LIN {X 0,Y 474.621,Z 246.364,A -85,B 0,C 180,E1 -7356.642,E2 -7356.642} C_VEL
LIN {X 0,Y 474.629,Z 246.359,A -85,B 0,C 180,E1 -7360.089,E2 -7360.089} C_VEL
LIN {X 0,Y 474.61,Z 246.369,A -85,B 0,C 180,E1 -7362.773,E2 -7362.773} C_VEL
LIN {X 0,Y 474.616,Z 246.361,A -85,B 0,C 180,E1 -7365.42,E2 -7365.42} C_VEL
LIN {X 0,Y 474.69,Z 246.352,A -85,B 0,C 180,E1 -7368.037,E2 -7368.037} C_VEL
LIN {X 0,Y 474.653,Z 246.356,A -85,B 0,C 180,E1 -7371.485,E2 -7371.485} C_VEL
LIN {X 0,Y 474.713,Z 246.35,A -85,B 0,C 180,E1 -7374.052,E2 -7374.052} C_VEL
LIN {X 0,Y 474.865,Z 246.329,A -85,B 0,C 180,E1 -7377.455,E2 -7377.455} C_VEL
LIN {X 0,Y 474.862,Z 246.332,A -85,B 0,C 180,E1 -7380,E2 -7380} C_VEL
LIN {X 0,Y 474.855,Z 246.338,A -85,B 0,C 180,E1 -7382.545,E2 -7382.545} C_VEL
LIN {X 0,Y 474.722,Z 246.349,A -85,B 0,C 180,E1 -7385.949,E2 -7385.949} C_VEL
LIN {X 0,Y 474.646,Z 246.363,A -85,B 0,C 180,E1 -7388.515,E2 -7388.515} C_VEL
LIN {X 0,Y 474.679,Z 246.356,A -85,B 0,C 180,E1 -7391.963,E2 -7391.963} C_VEL
LIN {X 0,Y 474.685,Z 246.352,A -85,B 0,C 180,E1 -7395.456,E2 -7395.456} C_VEL
LIN {X 0,Y 474.647,Z 246.356,A -85,B 0,C 180,E1 -7399.011,E2 -7399.011} C_VEL
LIN {X 0,Y 474.575,Z 246.368,A -85,B 0,C 180,E1 -7401.73,E2 -7401.73} C_VEL
LIN {X 0,Y 474.614,Z 246.364,A -85,B 0,C 180,E1 -7404.496,E2 -7404.496} C_VEL
LIN {X 0,Y 474.586,Z 246.364,A -85,B 0,C 180,E1 -7407.327,E2 -7407.327} C_VEL
LIN {X 0,Y 474.584,Z 246.369,A -85,B 0,C 180,E1 -7410.232,E2 -7410.232} C_VEL
LIN {X 0,Y 474.604,Z 246.362,A -85,B 0,C 180,E1 -7413.224,E2 -7413.224} C_VEL
LIN {X 0,Y 474.561,Z 246.37,A -85,B 0,C 180,E1 -7416.327,E2 -7416.327} C_VEL
LIN {X 0,Y 474.59,Z 246.367,A -85,B 0,C 180,E1 -7419.552,E2 -7419.552} C_VEL
LIN {X 0,Y 474.558,Z 246.367,A -85,B 0,C 180,E1 -7422.941,E2 -7422.941} C_VEL
LIN {X 0,Y 474.592,Z 246.369,A -85,B 0,C 180,E1 -7425.895,E2 -7425.895} C_VEL
LIN {X 0,Y 474.576,Z 246.366,A -85,B 0,C 180,E1 -7429.049,E2 -7429.049} C_VEL
LIN {X 0,Y 474.582,Z 246.372,A -85,B 0,C 180,E1 -7431.709,E2 -7431.709} C_VEL
LIN {X 0,Y 474.598,Z 246.362,A -85,B 0,C 180,E1 -7434.725,E2 -7434.725} C_VEL
LIN {X 0,Y 474.608,Z 246.366,A -85,B 0,C 180,E1 -7437.787,E2 -7437.787} C_VEL
LIN {X 0,Y 474.576,Z 246.366,A -85,B 0,C 180,E1 -7440.896,E2 -7440.896} C_VEL
LIN {X 0,Y 474.57,Z 246.372,A -85,B 0,C 180,E1 -7443.624,E2 -7443.624} C_VEL
LIN {X 0,Y 474.598,Z 246.363,A -85,B 0,C 180,E1 -7446.654,E2 -7446.654} C_VEL
LIN {X 0,Y 474.65,Z 246.362,A -85,B 0,C 180,E1 -7449.185,E2 -7449.185} C_VEL
LIN {X 0,Y 474.62,Z 246.363,A -85,B 0,C 180,E1 -7451.678,E2 -7451.678} C_VEL
LIN {X 0,Y 473.952,Z 246.443,A -85,B 0,C 180,E1 -7452.387,E2 -7452.387} C_VEL
LIN {X 0,Y 471.093,Z 246.804,A -85,B 0,C 180,E1 -7453.537,E2 -7453.537} C_VEL
LIN {X 0,Y 468.675,Z 247.109,A -85,B 0,C 180,E1 -7454.465,E2 -7454.465} C_VEL
LIN {X 0,Y 467.639,Z 247.236,A -85,B 0,C 180,E1 -7455.182,E2 -7455.182} C_VEL
LIN {X 0,Y 467.556,Z 247.244,A -85,B 0,C 180,E1 -7455.425,E2 -7455.425} C_VEL
LIN {X 0,Y 467.651,Z 247.231,A -85,B 0,C 180,E1 -7457.855,E2 -7457.855} C_VEL
LIN {X 0,Y 467.634,Z 247.345,A -85,B 0,C 180,E1 -7461.248,E2 -7461.248} C_VEL
LIN {X 0,Y 467.783,Z 248.185,A -85,B 0,C 180,E1 -7461.4,E2 -7461.4} C_VEL
LIN {X 0,Y 471.317,Z 258.187,A -85,B 0,C 180,E1 -7461.7,E2 -7461.7} C_VEL
LIN {X 0,Y 470.726,Z 335.625,A -85,B 0,C 180,E1 -7462.898,E2 -7462.898} C_VEL
LIN {X 0,Y 470.617,Z 348.645,A -85,B 0,C 180,E1 -7463.274,E2 -7463.274} C_VEL
LIN {X 0,Y 470.403,Z 361.714,A -85,B 0,C 180,E1 -7463.836,E2 -7463.836} C_VEL
LIN {X 0,Y 470.089,Z 373.512,A -85,B 0,C 180,E1 -7464.531,E2 -7464.531} C_VEL
LIN {X 0,Y 469.636,Z 384.793,A -85,B 0,C 180,E1 -7465.387,E2 -7465.387} C_VEL
LIN {X 0,Y 469.199,Z 394.954,A -85,B 0,C 180,E1 -7466.351,E2 -7466.351} C_VEL
LIN {X 0,Y 468.764,Z 404.111,A -85,B 0,C 180,E1 -7467.423,E2 -7467.423} C_VEL
LIN {X 0,Y 468.378,Z 412.945,A -85,B 0,C 180,E1 -7468.711,E2 -7468.711} C_VEL
LIN {X 0,Y 467.943,Z 420.099,A -85,B 0,C 180,E1 -7470,E2 -7470} C_VEL
LIN {X 0,Y 467.634,Z 425.83,A -85,B 0,C 180,E1 -7471.292,E2 -7471.292} C_VEL
LIN {X 0,Y 467.486,Z 430.339,A -85,B 0,C 180,E1 -7472.585,E2 -7472.585} C_VEL
LIN {X 0,Y 467.33,Z 432.748,A -85,B 0,C 180,E1 -7473.449,E2 -7473.449} C_VEL
LIN {X 0,Y 467.278,Z 436.248,A -85,B 0,C 180,E1 -7475.178,E2 -7475.178} C_VEL
LIN {X 0,Y 467.236,Z 437.399,A -85,B 0,C 180,E1 -7476.044,E2 -7476.044} C_VEL
LIN {X 0,Y 467.182,Z 438.465,A -85,B 0,C 180,E1 -7477.781,E2 -7477.781} C_VEL
LIN {X 0,Y 467.157,Z 438.436,A -85,B 0,C 180,E1 -7478.653,E2 -7478.653} C_VEL
LIN {X 0,Y 467.19,Z 438.007,A -85,B 0,C 180,E1 -7479.525,E2 -7479.525} C_VEL
LIN {X 0,Y 467.318,Z 435.892,A -85,B 0,C 180,E1 -7481.274,E2 -7481.274} C_VEL
LIN {X 0,Y 467.444,Z 433.216,A -85,B 0,C 180,E1 -7482.592,E2 -7482.592} C_VEL
LIN {X 0,Y 467.624,Z 429.5,A -85,B 0,C 180,E1 -7483.914,E2 -7483.914} C_VEL
LIN {X 0,Y 467.917,Z 424.627,A -85,B 0,C 180,E1 -7485.239,E2 -7485.239} C_VEL
LIN {X 0,Y 468.213,Z 418.444,A -85,B 0,C 180,E1 -7486.57,E2 -7486.57} C_VEL
LIN {X 0,Y 468.663,Z 410.633,A -85,B 0,C 180,E1 -7487.903,E2 -7487.903} C_VEL
LIN {X 0,Y 469.116,Z 402.581,A -85,B 0,C 180,E1 -7489.017,E2 -7489.017} C_VEL
LIN {X 0,Y 469.568,Z 392.679,A -85,B 0,C 180,E1 -7490.135,E2 -7490.135} C_VEL
LIN {X 0,Y 469.997,Z 382.87,A -85,B 0,C 180,E1 -7491.031,E2 -7491.031} C_VEL
LIN {X 0,Y 470.489,Z 372.14,A -85,B 0,C 180,E1 -7491.813,E2 -7491.813} C_VEL
LIN {X 0,Y 470.802,Z 360.376,A -85,B 0,C 180,E1 -7492.482,E2 -7492.482} C_VEL
LIN {X 0,Y 470.994,Z 347.261,A -85,B 0,C 180,E1 -7493.031,E2 -7493.031} C_VEL
LIN {X 0,Y 471.146,Z 334.596,A -85,B 0,C 180,E1 -7493.372,E2 -7493.372} C_VEL
LIN {X 0,Y 471.661,Z 258.296,A -85,B 0,C 180,E1 -7494.57,E2 -7494.57} C_VEL
LIN {X 0,Y 467.796,Z 248.157,A -85,B 0,C 180,E1 -7494.925,E2 -7494.925} C_VEL
LIN {X 0,Y 467.618,Z 247.318,A -85,B 0,C 180,E1 -7495.096,E2 -7495.096} C_VEL
LIN {X 0,Y 467.564,Z 247.242,A -85,B 0,C 180,E1 -7497.772,E2 -7497.772} C_VEL
LIN {X 0,Y 467.552,Z 247.228,A -85,B 0,C 180,E1 -7501.041,E2 -7501.041} C_VEL
LIN {X 0,Y 467.577,Z 247.243,A -85,B 0,C 180,E1 -7504.239,E2 -7504.239} C_VEL
LIN {X 0,Y 467.535,Z 247.227,A -85,B 0,C 180,E1 -7507.183,E2 -7507.183} C_VEL
LIN {X 0,Y 467.556,Z 247.246,A -85,B 0,C 180,E1 -7510.266,E2 -7510.266} C_VEL
LIN {X 0,Y 467.545,Z 247.243,A -85,B 0,C 180,E1 -7513.745,E2 -7513.745} C_VEL
LIN {X 0,Y 467.542,Z 247.241,A -85,B 0,C 180,E1 -7516.253,E2 -7516.253} C_VEL
LIN {X 0,Y 467.554,Z 247.242,A -85,B 0,C 180,E1 -7519.732,E2 -7519.732} C_VEL
LIN {X 0,Y 467.514,Z 247.239,A -85,B 0,C 180,E1 -7522.818,E2 -7522.818} C_VEL
LIN {X 0,Y 467.583,Z 247.24,A -85,B 0,C 180,E1 -7525.758,E2 -7525.758} C_VEL
LIN {X 0,Y 467.563,Z 247.226,A -85,B 0,C 180,E1 -7528.955,E2 -7528.955} C_VEL
LIN {X 0,Y 467.542,Z 247.245,A -85,B 0,C 180,E1 -7532.226,E2 -7532.226} C_VEL
LIN {X 0,Y 467.564,Z 247.238,A -85,B 0,C 180,E1 -7535.11,E2 -7535.11} C_VEL
LIN {X 0,Y 467.528,Z 247.228,A -85,B 0,C 180,E1 -7537.925,E2 -7537.925} C_VEL
LIN {X 0,Y 467.615,Z 247.23,A -85,B 0,C 180,E1 -7540.692,E2 -7540.692} C_VEL
LIN {X 0,Y 467.631,Z 247.23,A -85,B 0,C 180,E1 -7544.304,E2 -7544.304} C_VEL
LIN {X 0,Y 467.649,Z 247.235,A -85,B 0,C 180,E1 -7547.854,E2 -7547.854} C_VEL
LIN {X 0,Y 467.649,Z 247.224,A -85,B 0,C 180,E1 -7551.356,E2 -7551.356} C_VEL
LIN {X 0,Y 467.694,Z 247.227,A -85,B 0,C 180,E1 -7553.962,E2 -7553.962} C_VEL
LIN {X 0,Y 467.804,Z 247.209,A -85,B 0,C 180,E1 -7557.417,E2 -7557.417} C_VEL
LIN {X 0,Y 467.839,Z 247.206,A -85,B 0,C 180,E1 -7560,E2 -7560} C_VEL
LIN {X 0,Y 467.813,Z 247.204,A -85,B 0,C 180,E1 -7562.583,E2 -7562.583} C_VEL
LIN {X 0,Y 467.685,Z 247.223,A -85,B 0,C 180,E1 -7566.038,E2 -7566.038} C_VEL
LIN {X 0,Y 467.657,Z 247.224,A -85,B 0,C 180,E1 -7568.643,E2 -7568.643} C_VEL
LIN {X 0,Y 467.646,Z 247.225,A -85,B 0,C 180,E1 -7572.357,E2 -7572.357} C_VEL
LIN {X 0,Y 467.616,Z 247.235,A -85,B 0,C 180,E1 -7575.873,E2 -7575.873} C_VEL
LIN {X 0,Y 467.612,Z 247.239,A -85,B 0,C 180,E1 -7579.308,E2 -7579.308} C_VEL
LIN {X 0,Y 467.523,Z 247.242,A -85,B 0,C 180,E1 -7582.074,E2 -7582.074} C_VEL
LIN {X 0,Y 467.548,Z 247.246,A -85,B 0,C 180,E1 -7584.89,E2 -7584.89} C_VEL
LIN {X 0,Y 467.536,Z 247.235,A -85,B 0,C 180,E1 -7587.774,E2 -7587.774} C_VEL
LIN {X 0,Y 467.531,Z 247.251,A -85,B 0,C 180,E1 -7591.039,E2 -7591.039} C_VEL
LIN {X 0,Y 467.562,Z 247.232,A -85,B 0,C 180,E1 -7593.79,E2 -7593.79} C_VEL
LIN {X 0,Y 467.5,Z 247.254,A -85,B 0,C 180,E1 -7596.965,E2 -7596.965} C_VEL
LIN {X 0,Y 467.556,Z 247.24,A -85,B 0,C 180,E1 -7599.952,E2 -7599.952} C_VEL
LIN {X 0,Y 467.513,Z 247.25,A -85,B 0,C 180,E1 -7602.569,E2 -7602.569} C_VEL
LIN {X 0,Y 467.558,Z 247.245,A -85,B 0,C 180,E1 -7605.052,E2 -7605.052} C_VEL
LIN {X 0,Y 467.551,Z 247.245,A -85,B 0,C 180,E1 -7608.727,E2 -7608.727} C_VEL
LIN {X 0,Y 467.531,Z 247.242,A -85,B 0,C 180,E1 -7611.953,E2 -7611.953} C_VEL
LIN {X 0,Y 467.547,Z 247.237,A -85,B 0,C 180,E1 -7615.166,E2 -7615.166} C_VEL
LIN {X 0,Y 467.544,Z 247.239,A -85,B 0,C 180,E1 -7618.257,E2 -7618.257} C_VEL
LIN {X 0,Y 467.564,Z 247.452,A -85,B 0,C 180,E1 -7620.587,E2 -7620.587} C_VEL
LIN {X 0,Y 470.411,Z 260.504,A -85,B 0,C 180,E1 -7622.651,E2 -7622.651} C_VEL
LIN {X 0,Y 470.807,Z 263.899,A -85,B 0,C 180,E1 -7623.157,E2 -7623.157} C_VEL
LIN {X 0,Y 469.848,Z 285.592,A -85,B 0,C 180,E1 -7626.18,E2 -7626.18} C_VEL
LIN {X 0,Y 469.068,Z 307.215,A -85,B 0,C 180,E1 -7629.155,E2 -7629.155} C_VEL
LIN {X 0,Y 468.414,Z 328.784,A -85,B 0,C 180,E1 -7632.087,E2 -7632.087} C_VEL
LIN {X 0,Y 468.237,Z 334.47,A -85,B 0,C 180,E1 -7632.84,E2 -7632.84} C_VEL
LIN {X 0,Y 470.969,Z 358.48,A -85,B 0,C 180,E1 -7633.353,E2 -7633.353} C_VEL
LIN {X 0,Y 471.032,Z 374.98,A -85,B 0,C 180,E1 -7633.615,E2 -7633.615} C_VEL
LIN {X 0,Y 470.493,Z 444.897,A -85,B 0,C 180,E1 -7634.708,E2 -7634.708} C_VEL
LIN {X 0,Y 470.06,Z 458.205,A -85,B 0,C 180,E1 -7635.082,E2 -7635.082} C_VEL
LIN {X 0,Y 469.548,Z 470.424,A -85,B 0,C 180,E1 -7635.591,E2 -7635.591} C_VEL
LIN {X 0,Y 469.037,Z 481.969,A -85,B 0,C 180,E1 -7636.239,E2 -7636.239} C_VEL
LIN {X 0,Y 468.504,Z 492.547,A -85,B 0,C 180,E1 -7636.996,E2 -7636.996} C_VEL
LIN {X 0,Y 468.07,Z 503.465,A -85,B 0,C 180,E1 -7637.975,E2 -7637.975} C_VEL
LIN {X 0,Y 467.631,Z 512.407,A -85,B 0,C 180,E1 -7638.953,E2 -7638.953} C_VEL
LIN {X 0,Y 467.222,Z 522.165,A -85,B 0,C 180,E1 -7640.257,E2 -7640.257} C_VEL
LIN {X 0,Y 467.016,Z 529.966,A -85,B 0,C 180,E1 -7641.563,E2 -7641.563} C_VEL
LIN {X 0,Y 466.912,Z 537.197,A -85,B 0,C 180,E1 -7643.084,E2 -7643.084} C_VEL
LIN {X 0,Y 466.899,Z 542.022,A -85,B 0,C 180,E1 -7644.385,E2 -7644.385} C_VEL
LIN {X 0,Y 466.948,Z 545.721,A -85,B 0,C 180,E1 -7645.684,E2 -7645.684} C_VEL
LIN {X 0,Y 466.99,Z 547.631,A -85,B 0,C 180,E1 -7646.549,E2 -7646.549} C_VEL
LIN {X 0,Y 466.887,Z 550.075,A -85,B 0,C 180,E1 -7648.274,E2 -7648.274} C_VEL
LIN {X 0,Y 466.897,Z 550.703,A -85,B 0,C 180,E1 -7649.137,E2 -7649.137} C_VEL
LIN {X 0,Y 466.917,Z 550.927,A -85,B 0,C 180,E1 -7650,E2 -7650} C_VEL
LIN {X 0,Y 466.897,Z 550.703,A -85,B 0,C 180,E1 -7650.862,E2 -7650.862} C_VEL
LIN {X 0,Y 466.91,Z 549.066,A -85,B 0,C 180,E1 -7652.588,E2 -7652.588} C_VEL
LIN {X 0,Y 466.987,Z 547.639,A -85,B 0,C 180,E1 -7653.451,E2 -7653.451} C_VEL
LIN {X 0,Y 466.887,Z 544.613,A -85,B 0,C 180,E1 -7654.749,E2 -7654.749} C_VEL
LIN {X 0,Y 466.888,Z 539.767,A -85,B 0,C 180,E1 -7656.251,E2 -7656.251} C_VEL
LIN {X 0,Y 466.974,Z 533.211,A -85,B 0,C 180,E1 -7657.784,E2 -7657.784} C_VEL
LIN {X 0,Y 467.139,Z 526.131,A -85,B 0,C 180,E1 -7659.089,E2 -7659.089} C_VEL
LIN {X 0,Y 467.403,Z 517.268,A -85,B 0,C 180,E1 -7660.395,E2 -7660.395} C_VEL
LIN {X 0,Y 467.757,Z 507.203,A -85,B 0,C 180,E1 -7661.592,E2 -7661.592} C_VEL
LIN {X 0,Y 468.289,Z 497.301,A -85,B 0,C 180,E1 -7662.547,E2 -7662.547} C_VEL
LIN {X 0,Y 468.754,Z 485.756,A -85,B 0,C 180,E1 -7663.437,E2 -7663.437} C_VEL
LIN {X 0,Y 469.301,Z 473.12,A -85,B 0,C 180,E1 -7664.194,E2 -7664.194} C_VEL
LIN {X 0,Y 469.808,Z 460.235,A -85,B 0,C 180,E1 -7664.76,E2 -7664.76} C_VEL
LIN {X 0,Y 470.254,Z 446.5,A -85,B 0,C 180,E1 -7665.161,E2 -7665.161} C_VEL
LIN {X 0,Y 470.591,Z 400.642,A -85,B 0,C 180,E1 -7665.886,E2 -7665.886} C_VEL
LIN {X 0,Y 470.806,Z 359,A -85,B 0,C 180,E1 -7666.521,E2 -7666.521} C_VEL
LIN {X 0,Y 468.174,Z 335.117,A -85,B 0,C 180,E1 -7666.992,E2 -7666.992} C_VEL
LIN {X 0,Y 468.811,Z 312.964,A -85,B 0,C 180,E1 -7669.94,E2 -7669.94} C_VEL
LIN {X 0,Y 469.582,Z 287.643,A -85,B 0,C 180,E1 -7673.366,E2 -7673.366} C_VEL
LIN {X 0,Y 470.464,Z 263.767,A -85,B 0,C 180,E1 -7676.624,E2 -7676.624} C_VEL
LIN {X 0,Y 469.895,Z 258.487,A -85,B 0,C 180,E1 -7677.38,E2 -7677.38} C_VEL
LIN {X 0,Y 467.548,Z 247.389,A -85,B 0,C 180,E1 -7679.076,E2 -7679.076} C_VEL
LIN {X 0,Y 467.541,Z 247.249,A -85,B 0,C 180,E1 -7681.742,E2 -7681.742} C_VEL
LIN {X 0,Y 467.544,Z 247.245,A -85,B 0,C 180,E1 -7684.833,E2 -7684.833} C_VEL
LIN {X 0,Y 467.528,Z 247.244,A -85,B 0,C 180,E1 -7688.047,E2 -7688.047} C_VEL
LIN {X 0,Y 467.547,Z 247.248,A -85,B 0,C 180,E1 -7691.404,E2 -7691.404} C_VEL
LIN {X 0,Y 467.553,Z 247.245,A -85,B 0,C 180,E1 -7695.051,E2 -7695.051} C_VEL
LIN {X 0,Y 467.551,Z 247.243,A -85,B 0,C 180,E1 -7698.725,E2 -7698.725} C_VEL
LIN {X 0,Y 467.534,Z 247.243,A -85,B 0,C 180,E1 -7701.952,E2 -7701.952} C_VEL
LIN {X 0,Y 467.535,Z 247.249,A -85,B 0,C 180,E1 -7705.165,E2 -7705.165} C_VEL
LIN {X 0,Y 467.533,Z 247.243,A -85,B 0,C 180,E1 -7708.256,E2 -7708.256} C_VEL
LIN {X 0,Y 467.527,Z 247.248,A -85,B 0,C 180,E1 -7711.247,E2 -7711.247} C_VEL
LIN {X 0,Y 467.549,Z 247.242,A -85,B 0,C 180,E1 -7714.405,E2 -7714.405} C_VEL
LIN {X 0,Y 467.558,Z 247.246,A -85,B 0,C 180,E1 -7716.995,E2 -7716.995} C_VEL
LIN {X 0,Y 467.598,Z 247.234,A -85,B 0,C 180,E1 -7719.776,E2 -7719.776} C_VEL
LIN {X 0,Y 467.573,Z 247.242,A -85,B 0,C 180,E1 -7722.505,E2 -7722.505} C_VEL
LIN {X 0,Y 467.578,Z 247.239,A -85,B 0,C 180,E1 -7725.196,E2 -7725.196} C_VEL
LIN {X 0,Y 467.642,Z 247.229,A -85,B 0,C 180,E1 -7727.854,E2 -7727.854} C_VEL
LIN {X 0,Y 467.621,Z 247.232,A -85,B 0,C 180,E1 -7731.356,E2 -7731.356} C_VEL
LIN {X 0,Y 467.678,Z 247.225,A -85,B 0,C 180,E1 -7733.962,E2 -7733.962} C_VEL
LIN {X 0,Y 467.806,Z 247.208,A -85,B 0,C 180,E1 -7737.417,E2 -7737.417} C_VEL
LIN {X 0,Y 467.832,Z 247.207,A -85,B 0,C 180,E1 -7740,E2 -7740} C_VEL
LIN {X 0,Y 467.795,Z 247.216,A -85,B 0,C 180,E1 -7742.583,E2 -7742.583} C_VEL
LIN {X 0,Y 467.687,Z 247.227,A -85,B 0,C 180,E1 -7746.038,E2 -7746.038} C_VEL
LIN {X 0,Y 467.615,Z 247.237,A -85,B 0,C 180,E1 -7748.644,E2 -7748.644} C_VEL
LIN {X 0,Y 467.635,Z 247.237,A -85,B 0,C 180,E1 -7752.354,E2 -7752.354} C_VEL
LIN {X 0,Y 467.611,Z 247.236,A -85,B 0,C 180,E1 -7755.874,E2 -7755.874} C_VEL
LIN {X 0,Y 467.606,Z 247.233,A -85,B 0,C 180,E1 -7759.309,E2 -7759.309} C_VEL
LIN {X 0,Y 467.519,Z 247.252,A -85,B 0,C 180,E1 -7762.075,E2 -7762.075} C_VEL
LIN {X 0,Y 467.543,Z 247.241,A -85,B 0,C 180,E1 -7764.891,E2 -7764.891} C_VEL
LIN {X 0,Y 467.533,Z 247.247,A -85,B 0,C 180,E1 -7767.775,E2 -7767.775} C_VEL
LIN {X 0,Y 467.535,Z 247.242,A -85,B 0,C 180,E1 -7771.041,E2 -7771.041} C_VEL
LIN {X 0,Y 467.566,Z 247.242,A -85,B 0,C 180,E1 -7774.241,E2 -7774.241} C_VEL
LIN {X 0,Y 467.505,Z 247.247,A -85,B 0,C 180,E1 -7777.182,E2 -7777.182} C_VEL
LIN {X 0,Y 467.509,Z 247.248,A -85,B 0,C 180,E1 -7780.272,E2 -7780.272} C_VEL
LIN {X 0,Y 467.509,Z 247.246,A -85,B 0,C 180,E1 -7782.57,E2 -7782.57} C_VEL
LIN {X 0,Y 467.556,Z 247.24,A -85,B 0,C 180,E1 -7785.053,E2 -7785.053} C_VEL
LIN {X 0,Y 467.545,Z 247.241,A -85,B 0,C 180,E1 -7788.729,E2 -7788.729} C_VEL
LIN {X 0,Y 467.533,Z 247.246,A -85,B 0,C 180,E1 -7791.954,E2 -7791.954} C_VEL
LIN {X 0,Y 467.536,Z 247.245,A -85,B 0,C 180,E1 -7795.166,E2 -7795.166} C_VEL
LIN {X 0,Y 467.54,Z 247.242,A -85,B 0,C 180,E1 -7798.258,E2 -7798.258} C_VEL
LIN {X 0,Y 467.525,Z 247.248,A -85,B 0,C 180,E1 -7801.248,E2 -7801.248} C_VEL
LIN {X 0,Y 467.561,Z 247.239,A -85,B 0,C 180,E1 -7804.406,E2 -7804.406} C_VEL
LIN {X 0,Y 467.552,Z 247.243,A -85,B 0,C 180,E1 -7806.996,E2 -7806.996} C_VEL
LIN {X 0,Y 467.594,Z 247.238,A -85,B 0,C 180,E1 -7809.777,E2 -7809.777} C_VEL
LIN {X 0,Y 467.577,Z 247.237,A -85,B 0,C 180,E1 -7812.506,E2 -7812.506} C_VEL
LIN {X 0,Y 467.556,Z 247.244,A -85,B 0,C 180,E1 -7815.425,E2 -7815.425} C_VEL
LIN {X 0,Y 466.897,Z 247.323,A -85,B 0,C 180,E1 -7816.144,E2 -7816.144} C_VEL
LIN {X 0,Y 464.065,Z 247.682,A -85,B 0,C 180,E1 -7817.313,E2 -7817.313} C_VEL
LIN {X 0,Y 461.667,Z 247.978,A -85,B 0,C 180,E1 -7818.256,E2 -7818.256} C_VEL
LIN {X 0,Y 460.634,Z 248.109,A -85,B 0,C 180,E1 -7818.984,E2 -7818.984} C_VEL
LIN {X 0,Y 460.549,Z 248.116,A -85,B 0,C 180,E1 -7819.23,E2 -7819.23} C_VEL
LIN {X 0,Y 460.608,Z 248.343,A -85,B 0,C 180,E1 -7821.058,E2 -7821.058} C_VEL
LIN {X 0,Y 460.859,Z 249.412,A -85,B 0,C 180,E1 -7821.191,E2 -7821.191} C_VEL
LIN {X 0,Y 464.461,Z 259.967,A -85,B 0,C 180,E1 -7821.494,E2 -7821.494} C_VEL
LIN {X 0,Y 463.859,Z 337.152,A -85,B 0,C 180,E1 -7822.711,E2 -7822.711} C_VEL
LIN {X 0,Y 463.781,Z 350.665,A -85,B 0,C 180,E1 -7823.119,E2 -7823.119} C_VEL
LIN {X 0,Y 463.526,Z 362.345,A -85,B 0,C 180,E1 -7823.635,E2 -7823.635} C_VEL
LIN {X 0,Y 463.205,Z 374.206,A -85,B 0,C 180,E1 -7824.341,E2 -7824.341} C_VEL
LIN {X 0,Y 462.731,Z 385.516,A -85,B 0,C 180,E1 -7825.209,E2 -7825.209} C_VEL
LIN {X 0,Y 462.269,Z 395.701,A -85,B 0,C 180,E1 -7826.187,E2 -7826.187} C_VEL
LIN {X 0,Y 461.87,Z 404.033,A -85,B 0,C 180,E1 -7827.166,E2 -7827.166} C_VEL
LIN {X 0,Y 461.479,Z 411.725,A -85,B 0,C 180,E1 -7828.255,E2 -7828.255} C_VEL
LIN {X 0,Y 461.029,Z 419.262,A -85,B 0,C 180,E1 -7829.564,E2 -7829.564} C_VEL
LIN {X 0,Y 460.704,Z 425.308,A -85,B 0,C 180,E1 -7830.874,E2 -7830.874} C_VEL
LIN {X 0,Y 460.484,Z 430.114,A -85,B 0,C 180,E1 -7832.187,E2 -7832.187} C_VEL
LIN {X 0,Y 460.283,Z 433.835,A -85,B 0,C 180,E1 -7833.502,E2 -7833.502} C_VEL
LIN {X 0,Y 460.248,Z 435.748,A -85,B 0,C 180,E1 -7834.379,E2 -7834.379} C_VEL
LIN {X 0,Y 460.234,Z 437.259,A -85,B 0,C 180,E1 -7835.257,E2 -7835.257} C_VEL
LIN {X 0,Y 460.166,Z 438.963,A -85,B 0,C 180,E1 -7836.909,E2 -7836.909} C_VEL
LIN {X 0,Y 460.142,Z 439.334,A -85,B 0,C 180,E1 -7837.901,E2 -7837.901} C_VEL
LIN {X 0,Y 460.125,Z 439.267,A -85,B 0,C 180,E1 -7838.786,E2 -7838.786} C_VEL
LIN {X 0,Y 460.141,Z 438.769,A -85,B 0,C 180,E1 -7839.672,E2 -7839.672} C_VEL
LIN {X 0,Y 460.307,Z 436.579,A -85,B 0,C 180,E1 -7841.448,E2 -7841.448} C_VEL
LIN {X 0,Y 460.433,Z 433.827,A -85,B 0,C 180,E1 -7842.787,E2 -7842.787} C_VEL
LIN {X 0,Y 460.654,Z 430.029,A -85,B 0,C 180,E1 -7844.129,E2 -7844.129} C_VEL
LIN {X 0,Y 460.99,Z 425.067,A -85,B 0,C 180,E1 -7845.474,E2 -7845.474} C_VEL
LIN {X 0,Y 461.305,Z 418.775,A -85,B 0,C 180,E1 -7846.826,E2 -7846.826} C_VEL
LIN {X 0,Y 461.816,Z 410.809,A -85,B 0,C 180,E1 -7848.178,E2 -7848.178} C_VEL
LIN {X 0,Y 462.329,Z 402.049,A -85,B 0,C 180,E1 -7849.381,E2 -7849.381} C_VEL
LIN {X 0,Y 462.759,Z 392.55,A -85,B 0,C 180,E1 -7850.445,E2 -7850.445} C_VEL
LIN {X 0,Y 463.24,Z 382.457,A -85,B 0,C 180,E1 -7851.353,E2 -7851.353} C_VEL
LIN {X 0,Y 463.772,Z 371.385,A -85,B 0,C 180,E1 -7852.145,E2 -7852.145} C_VEL
LIN {X 0,Y 464.081,Z 359.466,A -85,B 0,C 180,E1 -7852.81,E2 -7852.81} C_VEL
LIN {X 0,Y 464.273,Z 346.755,A -85,B 0,C 180,E1 -7853.325,E2 -7853.325} C_VEL
LIN {X 0,Y 464.431,Z 333.014,A -85,B 0,C 180,E1 -7853.671,E2 -7853.671} C_VEL
LIN {X 0,Y 464.952,Z 259.822,A -85,B 0,C 180,E1 -7854.832,E2 -7854.832} C_VEL
LIN {X 0,Y 460.76,Z 249.177,A -85,B 0,C 180,E1 -7855.21,E2 -7855.21} C_VEL
LIN {X 0,Y 460.555,Z 248.238,A -85,B 0,C 180,E1 -7855.373,E2 -7855.373} C_VEL
LIN {X 0,Y 460.518,Z 248.119,A -85,B 0,C 180,E1 -7858.235,E2 -7858.235} C_VEL
LIN {X 0,Y 460.522,Z 248.104,A -85,B 0,C 180,E1 -7861.282,E2 -7861.282} C_VEL
LIN {X 0,Y 460.522,Z 248.116,A -85,B 0,C 180,E1 -7864.503,E2 -7864.503} C_VEL
LIN {X 0,Y 460.493,Z 248.11,A -85,B 0,C 180,E1 -7867.623,E2 -7867.623} C_VEL
LIN {X 0,Y 460.515,Z 248.117,A -85,B 0,C 180,E1 -7871.012,E2 -7871.012} C_VEL
LIN {X 0,Y 460.51,Z 248.125,A -85,B 0,C 180,E1 -7874.589,E2 -7874.589} C_VEL
LIN {X 0,Y 460.472,Z 248.118,A -85,B 0,C 180,E1 -7877.812,E2 -7877.812} C_VEL
LIN {X 0,Y 460.508,Z 248.123,A -85,B 0,C 180,E1 -7880.135,E2 -7880.135} C_VEL
LIN {X 0,Y 460.458,Z 248.117,A -85,B 0,C 180,E1 -7883.468,E2 -7883.468} C_VEL
LIN {X 0,Y 460.524,Z 248.118,A -85,B 0,C 180,E1 -7886.674,E2 -7886.674} C_VEL
LIN {X 0,Y 460.502,Z 248.105,A -85,B 0,C 180,E1 -7889.759,E2 -7889.759} C_VEL
LIN {X 0,Y 460.487,Z 248.124,A -85,B 0,C 180,E1 -7892.75,E2 -7892.75} C_VEL
LIN {X 0,Y 460.517,Z 248.118,A -85,B 0,C 180,E1 -7895.666,E2 -7895.666} C_VEL
LIN {X 0,Y 460.516,Z 248.101,A -85,B 0,C 180,E1 -7898.578,E2 -7898.578} C_VEL
LIN {X 0,Y 460.578,Z 248.107,A -85,B 0,C 180,E1 -7901.31,E2 -7901.31} C_VEL
LIN {X 0,Y 460.599,Z 248.11,A -85,B 0,C 180,E1 -7904.058,E2 -7904.058} C_VEL
LIN {X 0,Y 460.602,Z 248.11,A -85,B 0,C 180,E1 -7907.665,E2 -7907.665} C_VEL
LIN {X 0,Y 460.601,Z 248.101,A -85,B 0,C 180,E1 -7911.223,E2 -7911.223} C_VEL
LIN {X 0,Y 460.66,Z 248.104,A -85,B 0,C 180,E1 -7913.869,E2 -7913.869} C_VEL
LIN {X 0,Y 460.748,Z 248.087,A -85,B 0,C 180,E1 -7917.377,E2 -7917.377} C_VEL
LIN {X 0,Y 460.809,Z 248.082,A -85,B 0,C 180,E1 -7920,E2 -7920} C_VEL
LIN {X 0,Y 460.758,Z 248.083,A -85,B 0,C 180,E1 -7922.623,E2 -7922.623} C_VEL
LIN {X 0,Y 460.651,Z 248.098,A -85,B 0,C 180,E1 -7926.131,E2 -7926.131} C_VEL
LIN {X 0,Y 460.608,Z 248.103,A -85,B 0,C 180,E1 -7928.776,E2 -7928.776} C_VEL
LIN {X 0,Y 460.59,Z 248.104,A -85,B 0,C 180,E1 -7932.435,E2 -7932.435} C_VEL
LIN {X 0,Y 460.572,Z 248.112,A -85,B 0,C 180,E1 -7935.988,E2 -7935.988} C_VEL
LIN {X 0,Y 460.558,Z 248.112,A -85,B 0,C 180,E1 -7938.899,E2 -7938.899} C_VEL
LIN {X 0,Y 460.509,Z 248.12,A -85,B 0,C 180,E1 -7941.486,E2 -7941.486} C_VEL
LIN {X 0,Y 460.509,Z 248.119,A -85,B 0,C 180,E1 -7944.334,E2 -7944.334} C_VEL
LIN {X 0,Y 460.482,Z 248.114,A -85,B 0,C 180,E1 -7947.25,E2 -7947.25} C_VEL
LIN {X 0,Y 460.487,Z 248.121,A -85,B 0,C 180,E1 -7950.242,E2 -7950.242} C_VEL
LIN {X 0,Y 460.512,Z 248.112,A -85,B 0,C 180,E1 -7953.326,E2 -7953.326} C_VEL
LIN {X 0,Y 460.455,Z 248.128,A -85,B 0,C 180,E1 -7956.531,E2 -7956.531} C_VEL
LIN {X 0,Y 460.505,Z 248.118,A -85,B 0,C 180,E1 -7959.865,E2 -7959.865} C_VEL
LIN {X 0,Y 460.452,Z 248.126,A -85,B 0,C 180,E1 -7962.893,E2 -7962.893} C_VEL
LIN {X 0,Y 460.5,Z 248.119,A -85,B 0,C 180,E1 -7965.832,E2 -7965.832} C_VEL
LIN {X 0,Y 460.504,Z 248.119,A -85,B 0,C 180,E1 -7968.986,E2 -7968.986} C_VEL
LIN {X 0,Y 460.476,Z 248.124,A -85,B 0,C 180,E1 -7972.375,E2 -7972.375} C_VEL
LIN {X 0,Y 460.531,Z 248.114,A -85,B 0,C 180,E1 -7975.623,E2 -7975.623} C_VEL
LIN {X 0,Y 460.503,Z 248.12,A -85,B 0,C 180,E1 -7978.742,E2 -7978.742} C_VEL
LIN {X 0,Y 460.526,Z 248.315,A -85,B 0,C 180,E1 -7980.319,E2 -7980.319} C_VEL
LIN {X 0,Y 463.436,Z 261.52,A -85,B 0,C 180,E1 -7982.45,E2 -7982.45} C_VEL
LIN {X 0,Y 463.905,Z 264.918,A -85,B 0,C 180,E1 -7982.968,E2 -7982.968} C_VEL
LIN {X 0,Y 462.923,Z 286.594,A -85,B 0,C 180,E1 -7986.039,E2 -7986.039} C_VEL
LIN {X 0,Y 462.094,Z 308.192,A -85,B 0,C 180,E1 -7989.059,E2 -7989.059} C_VEL
LIN {X 0,Y 461.316,Z 331.385,A -85,B 0,C 180,E1 -7992.26,E2 -7992.26} C_VEL
LIN {X 0,Y 461.279,Z 333.981,A -85,B 0,C 180,E1 -7992.568,E2 -7992.568} C_VEL
LIN {X 0,Y 464.071,Z 357.869,A -85,B 0,C 180,E1 -7993.076,E2 -7993.076} C_VEL
LIN {X 0,Y 464.375,Z 364.598,A -85,B 0,C 180,E1 -7993.195,E2 -7993.195} C_VEL
LIN {X 0,Y 463.652,Z 444.972,A -85,B 0,C 180,E1 -7994.477,E2 -7994.477} C_VEL
LIN {X 0,Y 463.178,Z 458.722,A -85,B 0,C 180,E1 -7994.883,E2 -7994.883} C_VEL
LIN {X 0,Y 462.668,Z 470.01,A -85,B 0,C 180,E1 -7995.372,E2 -7995.372} C_VEL
LIN {X 0,Y 462.121,Z 481.434,A -85,B 0,C 180,E1 -7996.029,E2 -7996.029} C_VEL
LIN {X 0,Y 461.47,Z 493.521,A -85,B 0,C 180,E1 -7996.931,E2 -7996.931} C_VEL
LIN {X 0,Y 461.023,Z 503.875,A -85,B 0,C 180,E1 -7997.9,E2 -7997.9} C_VEL
LIN {X 0,Y 460.517,Z 513.5,A -85,B 0,C 180,E1 -7999.003,E2 -7999.003} C_VEL
LIN {X 0,Y 460.104,Z 522.802,A -85,B 0,C 180,E1 -8000.327,E2 -8000.327} C_VEL
LIN {X 0,Y 459.931,Z 530.333,A -85,B 0,C 180,E1 -8001.653,E2 -8001.653} C_VEL
LIN {X 0,Y 459.845,Z 536.404,A -85,B 0,C 180,E1 -8002.977,E2 -8002.977} C_VEL
LIN {X 0,Y 459.829,Z 541.214,A -85,B 0,C 180,E1 -8004.298,E2 -8004.298} C_VEL
LIN {X 0,Y 459.888,Z 544.902,A -85,B 0,C 180,E1 -8005.617,E2 -8005.617} C_VEL
LIN {X 0,Y 459.941,Z 546.804,A -85,B 0,C 180,E1 -8006.496,E2 -8006.496} C_VEL
LIN {X 0,Y 459.832,Z 549.237,A -85,B 0,C 180,E1 -8008.248,E2 -8008.248} C_VEL
LIN {X 0,Y 459.844,Z 549.861,A -85,B 0,C 180,E1 -8009.124,E2 -8009.124} C_VEL
LIN {X 0,Y 459.868,Z 550.077,A -85,B 0,C 180,E1 -8010,E2 -8010} C_VEL
LIN {X 0,Y 459.846,Z 549.847,A -85,B 0,C 180,E1 -8010.875,E2 -8010.875} C_VEL
LIN {X 0,Y 459.856,Z 548.199,A -85,B 0,C 180,E1 -8012.627,E2 -8012.627} C_VEL
LIN {X 0,Y 459.939,Z 546.762,A -85,B 0,C 180,E1 -8013.504,E2 -8013.504} C_VEL
LIN {X 0,Y 459.818,Z 543.722,A -85,B 0,C 180,E1 -8014.822,E2 -8014.822} C_VEL
LIN {X 0,Y 459.82,Z 539.622,A -85,B 0,C 180,E1 -8016.141,E2 -8016.141} C_VEL
LIN {X 0,Y 459.884,Z 533.312,A -85,B 0,C 180,E1 -8017.684,E2 -8017.684} C_VEL
LIN {X 0,Y 460.026,Z 526.439,A -85,B 0,C 180,E1 -8019.009,E2 -8019.009} C_VEL
LIN {X 0,Y 460.284,Z 517.921,A -85,B 0,C 180,E1 -8020.335,E2 -8020.335} C_VEL
LIN {X 0,Y 460.643,Z 509.162,A -85,B 0,C 180,E1 -8021.439,E2 -8021.439} C_VEL
LIN {X 0,Y 461.176,Z 499.076,A -85,B 0,C 180,E1 -8022.478,E2 -8022.478} C_VEL
LIN {X 0,Y 461.644,Z 487.714,A -85,B 0,C 180,E1 -8023.424,E2 -8023.424} C_VEL
LIN {X 0,Y 462.199,Z 475.906,A -85,B 0,C 180,E1 -8024.192,E2 -8024.192} C_VEL
LIN {X 0,Y 462.718,Z 463.65,A -85,B 0,C 180,E1 -8024.794,E2 -8024.794} C_VEL
LIN {X 0,Y 463.214,Z 450.306,A -85,B 0,C 180,E1 -8025.256,E2 -8025.256} C_VEL
LIN {X 0,Y 463.489,Z 437.174,A -85,B 0,C 180,E1 -8025.528,E2 -8025.528} C_VEL
LIN {X 0,Y 463.894,Z 359.502,A -85,B 0,C 180,E1 -8026.729,E2 -8026.729} C_VEL
LIN {X 0,Y 461.147,Z 334.178,A -85,B 0,C 180,E1 -8027.242,E2 -8027.242} C_VEL
LIN {X 0,Y 461.793,Z 313.586,A -85,B 0,C 180,E1 -8030.024,E2 -8030.024} C_VEL
LIN {X 0,Y 462.592,Z 288.255,A -85,B 0,C 180,E1 -8033.503,E2 -8033.503} C_VEL
LIN {X 0,Y 463.517,Z 264.949,A -85,B 0,C 180,E1 -8036.728,E2 -8036.728} C_VEL
LIN {X 0,Y 463.161,Z 260.839,A -85,B 0,C 180,E1 -8037.322,E2 -8037.322} C_VEL
LIN {X 0,Y 460.509,Z 248.297,A -85,B 0,C 180,E1 -8039.26,E2 -8039.26} C_VEL
LIN {X 0,Y 460.507,Z 248.121,A -85,B 0,C 180,E1 -8042.285,E2 -8042.285} C_VEL
LIN {X 0,Y 460.494,Z 248.127,A -85,B 0,C 180,E1 -8045.446,E2 -8045.446} C_VEL
LIN {X 0,Y 460.474,Z 248.124,A -85,B 0,C 180,E1 -8048.887,E2 -8048.887} C_VEL
LIN {X 0,Y 460.491,Z 248.124,A -85,B 0,C 180,E1 -8051.597,E2 -8051.597} C_VEL
LIN {X 0,Y 460.502,Z 248.119,A -85,B 0,C 180,E1 -8054.589,E2 -8054.589} C_VEL
LIN {X 0,Y 460.465,Z 248.124,A -85,B 0,C 180,E1 -8057.812,E2 -8057.812} C_VEL
LIN {X 0,Y 460.5,Z 248.118,A -85,B 0,C 180,E1 -8060.134,E2 -8060.134} C_VEL
LIN {X 0,Y 460.45,Z 248.128,A -85,B 0,C 180,E1 -8063.468,E2 -8063.468} C_VEL
LIN {X 0,Y 460.489,Z 248.123,A -85,B 0,C 180,E1 -8066.672,E2 -8066.672} C_VEL
LIN {X 0,Y 460.481,Z 248.121,A -85,B 0,C 180,E1 -8069.758,E2 -8069.758} C_VEL
LIN {X 0,Y 460.473,Z 248.127,A -85,B 0,C 180,E1 -8072.75,E2 -8072.75} C_VEL
LIN {X 0,Y 460.5,Z 248.119,A -85,B 0,C 180,E1 -8075.665,E2 -8075.665} C_VEL
LIN {X 0,Y 460.506,Z 248.122,A -85,B 0,C 180,E1 -8078.579,E2 -8078.579} C_VEL
LIN {X 0,Y 460.569,Z 248.112,A -85,B 0,C 180,E1 -8081.31,E2 -8081.31} C_VEL
LIN {X 0,Y 460.573,Z 248.11,A -85,B 0,C 180,E1 -8084.058,E2 -8084.058} C_VEL
LIN {X 0,Y 460.596,Z 248.107,A -85,B 0,C 180,E1 -8087.666,E2 -8087.666} C_VEL
LIN {X 0,Y 460.576,Z 248.111,A -85,B 0,C 180,E1 -8091.223,E2 -8091.223} C_VEL
LIN {X 0,Y 460.645,Z 248.101,A -85,B 0,C 180,E1 -8093.869,E2 -8093.869} C_VEL
LIN {X 0,Y 460.751,Z 248.088,A -85,B 0,C 180,E1 -8097.377,E2 -8097.377} C_VEL
LIN {X 0,Y 460.781,Z 248.086,A -85,B 0,C 180,E1 -8100,E2 -8100} C_VEL
LIN {X 0,Y 460.739,Z 248.095,A -85,B 0,C 180,E1 -8102.623,E2 -8102.623} C_VEL
LIN {X 0,Y 460.653,Z 248.104,A -85,B 0,C 180,E1 -8106.131,E2 -8106.131} C_VEL
LIN {X 0,Y 460.57,Z 248.113,A -85,B 0,C 180,E1 -8108.777,E2 -8108.777} C_VEL
LIN {X 0,Y 460.585,Z 248.114,A -85,B 0,C 180,E1 -8112.436,E2 -8112.436} C_VEL
LIN {X 0,Y 460.567,Z 248.115,A -85,B 0,C 180,E1 -8115.989,E2 -8115.989} C_VEL
LIN {X 0,Y 460.553,Z 248.113,A -85,B 0,C 180,E1 -8118.9,E2 -8118.9} C_VEL
LIN {X 0,Y 460.505,Z 248.119,A -85,B 0,C 180,E1 -8121.487,E2 -8121.487} C_VEL
LIN {X 0,Y 460.504,Z 248.123,A -85,B 0,C 180,E1 -8124.335,E2 -8124.335} C_VEL
LIN {X 0,Y 460.477,Z 248.122,A -85,B 0,C 180,E1 -8127.25,E2 -8127.25} C_VEL
LIN {X 0,Y 460.491,Z 248.125,A -85,B 0,C 180,E1 -8130.242,E2 -8130.242} C_VEL
LIN {X 0,Y 460.506,Z 248.119,A -85,B 0,C 180,E1 -8133.327,E2 -8133.327} C_VEL
LIN {X 0,Y 460.449,Z 248.126,A -85,B 0,C 180,E1 -8136.532,E2 -8136.532} C_VEL
LIN {X 0,Y 460.485,Z 248.129,A -85,B 0,C 180,E1 -8139.868,E2 -8139.868} C_VEL
LIN {X 0,Y 460.452,Z 248.125,A -85,B 0,C 180,E1 -8142.894,E2 -8142.894} C_VEL
LIN {X 0,Y 460.489,Z 248.127,A -85,B 0,C 180,E1 -8145.834,E2 -8145.834} C_VEL
LIN {X 0,Y 460.499,Z 248.119,A -85,B 0,C 180,E1 -8148.987,E2 -8148.987} C_VEL
LIN {X 0,Y 460.477,Z 248.122,A -85,B 0,C 180,E1 -8152.376,E2 -8152.376} C_VEL
LIN {X 0,Y 460.518,Z 248.124,A -85,B 0,C 180,E1 -8155.623,E2 -8155.623} C_VEL
LIN {X 0,Y 460.503,Z 248.119,A -85,B 0,C 180,E1 -8158.743,E2 -8158.743} C_VEL
LIN {X 0,Y 460.495,Z 248.124,A -85,B 0,C 180,E1 -8161.764,E2 -8161.764} C_VEL
LIN {X 0,Y 460.509,Z 248.118,A -85,B 0,C 180,E1 -8164.704,E2 -8164.704} C_VEL
LIN {X 0,Y 460.497,Z 248.125,A -85,B 0,C 180,E1 -8167.572,E2 -8167.572} C_VEL
LIN {X 0,Y 460.522,Z 248.116,A -85,B 0,C 180,E1 -8170.383,E2 -8170.383} C_VEL
LIN {X 0,Y 460.54,Z 248.12,A -85,B 0,C 180,E1 -8173.146,E2 -8173.146} C_VEL
LIN {X 0,Y 460.521,Z 248.117,A -85,B 0,C 180,E1 -8175.868,E2 -8175.868} C_VEL
LIN {X 0,Y 460.595,Z 248.11,A -85,B 0,C 180,E1 -8178.56,E2 -8178.56} C_VEL
LIN {X 0,Y 460.549,Z 248.116,A -85,B 0,C 180,E1 -8179.23,E2 -8179.23} C_VEL
LIN {X 0,Y 460.404,Z 248.859,A -85,B 0,C 180,E1 -8179.684,E2 -8179.684} C_VEL
LIN {X 0,Y 460.073,Z 250.692,A -85,B 0,C 180,E1 -8180.092,E2 -8180.092} C_VEL
LIN {X 0,Y 459.632,Z 253.277,A -85,B 0,C 180,E1 -8180.45,E2 -8180.45} C_VEL
LIN {X 0,Y 458.887,Z 258.12,A -85,B 0,C 180,E1 -8180.878,E2 -8180.878} C_VEL
LIN {X 0,Y 457.95,Z 265.801,A -85,B 0,C 180,E1 -8181.284,E2 -8181.284} C_VEL
LIN {X 0,Y 457.573,Z 271.953,A -85,B 0,C 180,E1 -8181.444,E2 -8181.444} C_VEL
LIN {X 0,Y 457.01,Z 337.474,A -85,B 0,C 180,E1 -8182.49,E2 -8182.49} C_VEL
LIN {X 0,Y 456.876,Z 350.445,A -85,B 0,C 180,E1 -8182.876,E2 -8182.876} C_VEL
LIN {X 0,Y 456.651,Z 362.935,A -85,B 0,C 180,E1 -8183.428,E2 -8183.428} C_VEL
LIN {X 0,Y 456.322,Z 374.87,A -85,B 0,C 180,E1 -8184.144,E2 -8184.144} C_VEL
LIN {X 0,Y 455.828,Z 386.215,A -85,B 0,C 180,E1 -8185.025,E2 -8185.025} C_VEL
LIN {X 0,Y 455.341,Z 396.428,A -85,B 0,C 180,E1 -8186.018,E2 -8186.018} C_VEL
LIN {X 0,Y 454.867,Z 405.636,A -85,B 0,C 180,E1 -8187.122,E2 -8187.122} C_VEL
LIN {X 0,Y 454.425,Z 414.506,A -85,B 0,C 180,E1 -8188.45,E2 -8188.45} C_VEL
LIN {X 0,Y 453.942,Z 421.688,A -85,B 0,C 180,E1 -8189.779,E2 -8189.779} C_VEL
LIN {X 0,Y 453.581,Z 428.267,A -85,B 0,C 180,E1 -8191.332,E2 -8191.332} C_VEL
LIN {X 0,Y 453.384,Z 432.612,A -85,B 0,C 180,E1 -8192.666,E2 -8192.666} C_VEL
LIN {X 0,Y 453.237,Z 434.918,A -85,B 0,C 180,E1 -8193.556,E2 -8193.556} C_VEL
LIN {X 0,Y 453.213,Z 436.792,A -85,B 0,C 180,E1 -8194.447,E2 -8194.447} C_VEL
LIN {X 0,Y 453.19,Z 438.248,A -85,B 0,C 180,E1 -8195.339,E2 -8195.339} C_VEL
LIN {X 0,Y 453.124,Z 439.926,A -85,B 0,C 180,E1 -8197.128,E2 -8197.128} C_VEL
LIN {X 0,Y 453.099,Z 440.203,A -85,B 0,C 180,E1 -8198.025,E2 -8198.025} C_VEL
LIN {X 0,Y 453.101,Z 440.076,A -85,B 0,C 180,E1 -8198.923,E2 -8198.923} C_VEL
LIN {X 0,Y 453.147,Z 438.602,A -85,B 0,C 180,E1 -8200.726,E2 -8200.726} C_VEL
LIN {X 0,Y 453.367,Z 435.767,A -85,B 0,C 180,E1 -8202.413,E2 -8202.413} C_VEL
LIN {X 0,Y 453.623,Z 431.973,A -85,B 0,C 180,E1 -8203.895,E2 -8203.895} C_VEL
LIN {X 0,Y 453.9,Z 427.32,A -85,B 0,C 180,E1 -8205.261,E2 -8205.261} C_VEL
LIN {X 0,Y 454.324,Z 420.32,A -85,B 0,C 180,E1 -8206.849,E2 -8206.849} C_VEL
LIN {X 0,Y 454.858,Z 412.493,A -85,B 0,C 180,E1 -8208.233,E2 -8208.233} C_VEL
LIN {X 0,Y 455.423,Z 403.962,A -85,B 0,C 180,E1 -8209.445,E2 -8209.445} C_VEL
LIN {X 0,Y 455.904,Z 394.623,A -85,B 0,C 180,E1 -8210.53,E2 -8210.53} C_VEL
LIN {X 0,Y 456.38,Z 384.873,A -85,B 0,C 180,E1 -8211.453,E2 -8211.453} C_VEL
LIN {X 0,Y 456.901,Z 374.253,A -85,B 0,C 180,E1 -8212.258,E2 -8212.258} C_VEL
LIN {X 0,Y 457.309,Z 362.221,A -85,B 0,C 180,E1 -8212.965,E2 -8212.965} C_VEL
LIN {X 0,Y 457.513,Z 348.915,A -85,B 0,C 180,E1 -8213.54,E2 -8213.54} C_VEL
LIN {X 0,Y 457.649,Z 336.163,A -85,B 0,C 180,E1 -8213.893,E2 -8213.893} C_VEL
LIN {X 0,Y 458.226,Z 261.353,A -85,B 0,C 180,E1 -8215.103,E2 -8215.103} C_VEL
LIN {X 0,Y 453.709,Z 249.976,A -85,B 0,C 180,E1 -8215.521,E2 -8215.521} C_VEL
LIN {X 0,Y 453.51,Z 249.101,A -85,B 0,C 180,E1 -8215.688,E2 -8215.688} C_VEL
LIN {X 0,Y 453.47,Z 249,A -85,B 0,C 180,E1 -8218.714,E2 -8218.714} C_VEL
LIN {X 0,Y 453.462,Z 248.986,A -85,B 0,C 180,E1 -8221.799,E2 -8221.799} C_VEL
LIN {X 0,Y 453.476,Z 248.986,A -85,B 0,C 180,E1 -8224.989,E2 -8224.989} C_VEL
LIN {X 0,Y 453.452,Z 248.99,A -85,B 0,C 180,E1 -8228.312,E2 -8228.312} C_VEL
LIN {X 0,Y 453.47,Z 249,A -85,B 0,C 180,E1 -8230.611,E2 -8230.611} C_VEL
LIN {X 0,Y 453.458,Z 249.002,A -85,B 0,C 180,E1 -8234.221,E2 -8234.221} C_VEL
LIN {X 0,Y 453.419,Z 248.996,A -85,B 0,C 180,E1 -8236.999,E2 -8236.999} C_VEL
LIN {X 0,Y 453.468,Z 248.996,A -85,B 0,C 180,E1 -8239.412,E2 -8239.412} C_VEL
LIN {X 0,Y 453.433,Z 248.991,A -85,B 0,C 180,E1 -8242.808,E2 -8242.808} C_VEL
LIN {X 0,Y 453.471,Z 249.001,A -85,B 0,C 180,E1 -8246.086,E2 -8246.086} C_VEL
LIN {X 0,Y 453.471,Z 248.979,A -85,B 0,C 180,E1 -8249.24,E2 -8249.24} C_VEL
LIN {X 0,Y 453.47,Z 248.999,A -85,B 0,C 180,E1 -8252.293,E2 -8252.293} C_VEL
LIN {X 0,Y 453.486,Z 248.992,A -85,B 0,C 180,E1 -8255.264,E2 -8255.264} C_VEL
LIN {X 0,Y 453.475,Z 248.976,A -85,B 0,C 180,E1 -8258.415,E2 -8258.415} C_VEL
LIN {X 0,Y 453.517,Z 248.985,A -85,B 0,C 180,E1 -8261.008,E2 -8261.008} C_VEL
LIN {X 0,Y 453.563,Z 248.989,A -85,B 0,C 180,E1 -8263.879,E2 -8263.879} C_VEL
LIN {X 0,Y 453.558,Z 248.985,A -85,B 0,C 180,E1 -8267.471,E2 -8267.471} C_VEL
LIN {X 0,Y 453.569,Z 248.976,A -85,B 0,C 180,E1 -8271.086,E2 -8271.086} C_VEL
LIN {X 0,Y 453.628,Z 248.982,A -85,B 0,C 180,E1 -8273.774,E2 -8273.774} C_VEL
LIN {X 0,Y 453.695,Z 248.965,A -85,B 0,C 180,E1 -8277.336,E2 -8277.336} C_VEL
LIN {X 0,Y 453.758,Z 248.96,A -85,B 0,C 180,E1 -8280,E2 -8280} C_VEL
LIN {X 0,Y 453.705,Z 248.961,A -85,B 0,C 180,E1 -8282.663,E2 -8282.663} C_VEL
LIN {X 0,Y 453.62,Z 248.974,A -85,B 0,C 180,E1 -8286.226,E2 -8286.226} C_VEL
LIN {X 0,Y 453.574,Z 248.98,A -85,B 0,C 180,E1 -8288.914,E2 -8288.914} C_VEL
LIN {X 0,Y 453.557,Z 248.98,A -85,B 0,C 180,E1 -8292.529,E2 -8292.529} C_VEL
LIN {X 0,Y 453.531,Z 248.988,A -85,B 0,C 180,E1 -8296.196,E2 -8296.196} C_VEL
LIN {X 0,Y 453.51,Z 248.991,A -85,B 0,C 180,E1 -8299.039,E2 -8299.039} C_VEL
LIN {X 0,Y 453.469,Z 248.994,A -85,B 0,C 180,E1 -8301.836,E2 -8301.836} C_VEL
LIN {X 0,Y 453.461,Z 249,A -85,B 0,C 180,E1 -8304.737,E2 -8304.737} C_VEL
LIN {X 0,Y 453.454,Z 248.988,A -85,B 0,C 180,E1 -8307.942,E2 -8307.942} C_VEL
LIN {X 0,Y 453.447,Z 249.002,A -85,B 0,C 180,E1 -8310.762,E2 -8310.762} C_VEL
LIN {X 0,Y 453.46,Z 248.988,A -85,B 0,C 180,E1 -8313.914,E2 -8313.914} C_VEL
LIN {X 0,Y 453.43,Z 249.003,A -85,B 0,C 180,E1 -8317.192,E2 -8317.192} C_VEL
LIN {X 0,Y 453.465,Z 248.999,A -85,B 0,C 180,E1 -8320.612,E2 -8320.612} C_VEL
LIN {X 0,Y 453.476,Z 248.997,A -85,B 0,C 180,E1 -8324.529,E2 -8324.529} C_VEL
LIN {X 0,Y 453.429,Z 249.003,A -85,B 0,C 180,E1 -8328.072,E2 -8328.072} C_VEL
LIN {X 0,Y 453.424,Z 248.991,A -85,B 0,C 180,E1 -8330.804,E2 -8330.804} C_VEL
LIN {X 0,Y 453.437,Z 249.003,A -85,B 0,C 180,E1 -8333.916,E2 -8333.916} C_VEL
LIN {X 0,Y 453.478,Z 248.998,A -85,B 0,C 180,E1 -8336.814,E2 -8336.814} C_VEL
LIN {X 0,Y 453.466,Z 249.174,A -85,B 0,C 180,E1 -8340.038,E2 -8340.038} C_VEL
LIN {X 0,Y 456.46,Z 262.628,A -85,B 0,C 180,E1 -8342.254,E2 -8342.254} C_VEL
LIN {X 0,Y 457.02,Z 267.059,A -85,B 0,C 180,E1 -8342.938,E2 -8342.938} C_VEL
LIN {X 0,Y 455.93,Z 289.269,A -85,B 0,C 180,E1 -8346.132,E2 -8346.132} C_VEL
LIN {X 0,Y 455.069,Z 310.839,A -85,B 0,C 180,E1 -8349.194,E2 -8349.194} C_VEL
LIN {X 0,Y 454.289,Z 332.68,A -85,B 0,C 180,E1 -8352.238,E2 -8352.238} C_VEL
LIN {X 0,Y 456.427,Z 349.852,A -85,B 0,C 180,E1 -8352.638,E2 -8352.638} C_VEL
LIN {X 0,Y 457.657,Z 362.97,A -85,B 0,C 180,E1 -8352.902,E2 -8352.902} C_VEL
LIN {X 0,Y 456.885,Z 444.014,A -85,B 0,C 180,E1 -8354.212,E2 -8354.212} C_VEL
LIN {X 0,Y 456.323,Z 457.786,A -85,B 0,C 180,E1 -8354.622,E2 -8354.622} C_VEL
LIN {X 0,Y 455.771,Z 469.649,A -85,B 0,C 180,E1 -8355.146,E2 -8355.146} C_VEL
LIN {X 0,Y 455.185,Z 480.925,A -85,B 0,C 180,E1 -8355.812,E2 -8355.812} C_VEL
LIN {X 0,Y 454.581,Z 491.336,A -85,B 0,C 180,E1 -8356.591,E2 -8356.591} C_VEL
LIN {X 0,Y 454.128,Z 502.152,A -85,B 0,C 180,E1 -8357.6,E2 -8357.6} C_VEL
LIN {X 0,Y 453.571,Z 511.007,A -85,B 0,C 180,E1 -8358.606,E2 -8358.606} C_VEL
LIN {X 0,Y 453.193,Z 519.197,A -85,B 0,C 180,E1 -8359.727,E2 -8359.727} C_VEL
LIN {X 0,Y 452.922,Z 527.275,A -85,B 0,C 180,E1 -8361.073,E2 -8361.073} C_VEL
LIN {X 0,Y 452.807,Z 533.763,A -85,B 0,C 180,E1 -8362.419,E2 -8362.419} C_VEL
LIN {X 0,Y 452.711,Z 538.941,A -85,B 0,C 180,E1 -8363.761,E2 -8363.761} C_VEL
LIN {X 0,Y 452.716,Z 542.977,A -85,B 0,C 180,E1 -8365.102,E2 -8365.102} C_VEL
LIN {X 0,Y 452.876,Z 545.98,A -85,B 0,C 180,E1 -8366.441,E2 -8366.441} C_VEL
LIN {X 0,Y 452.776,Z 548.402,A -85,B 0,C 180,E1 -8368.221,E2 -8368.221} C_VEL
LIN {X 0,Y 452.791,Z 549.021,A -85,B 0,C 180,E1 -8369.11,E2 -8369.11} C_VEL
LIN {X 0,Y 452.82,Z 549.226,A -85,B 0,C 180,E1 -8370,E2 -8370} C_VEL
LIN {X 0,Y 452.795,Z 548.988,A -85,B 0,C 180,E1 -8370.889,E2 -8370.889} C_VEL
LIN {X 0,Y 452.803,Z 547.327,A -85,B 0,C 180,E1 -8372.668,E2 -8372.668} C_VEL
LIN {X 0,Y 452.891,Z 545.878,A -85,B 0,C 180,E1 -8373.558,E2 -8373.558} C_VEL
LIN {X 0,Y 452.753,Z 542.822,A -85,B 0,C 180,E1 -8374.897,E2 -8374.897} C_VEL
LIN {X 0,Y 452.765,Z 538.705,A -85,B 0,C 180,E1 -8376.237,E2 -8376.237} C_VEL
LIN {X 0,Y 452.806,Z 532.364,A -85,B 0,C 180,E1 -8377.805,E2 -8377.805} C_VEL
LIN {X 0,Y 452.977,Z 525.469,A -85,B 0,C 180,E1 -8379.15,E2 -8379.15} C_VEL
LIN {X 0,Y 453.256,Z 516.913,A -85,B 0,C 180,E1 -8380.497,E2 -8380.497} C_VEL
LIN {X 0,Y 453.583,Z 508.102,A -85,B 0,C 180,E1 -8381.62,E2 -8381.62} C_VEL
LIN {X 0,Y 454.175,Z 497.478,A -85,B 0,C 180,E1 -8382.721,E2 -8382.721} C_VEL
LIN {X 0,Y 454.69,Z 486.558,A -85,B 0,C 180,E1 -8383.633,E2 -8383.633} C_VEL
LIN {X 0,Y 455.267,Z 474.622,A -85,B 0,C 180,E1 -8384.413,E2 -8384.413} C_VEL
LIN {X 0,Y 455.828,Z 462.23,A -85,B 0,C 180,E1 -8385.023,E2 -8385.023} C_VEL
LIN {X 0,Y 456.305,Z 449.567,A -85,B 0,C 180,E1 -8385.464,E2 -8385.464} C_VEL
LIN {X 0,Y 456.604,Z 436.532,A -85,B 0,C 180,E1 -8385.74,E2 -8385.74} C_VEL
LIN {X 0,Y 457.001,Z 359.914,A -85,B 0,C 180,E1 -8386.943,E2 -8386.943} C_VEL
LIN {X 0,Y 454.107,Z 333.265,A -85,B 0,C 180,E1 -8387.492,E2 -8387.492} C_VEL
LIN {X 0,Y 454.751,Z 314.191,A -85,B 0,C 180,E1 -8390.112,E2 -8390.112} C_VEL
LIN {X 0,Y 455.606,Z 288.852,A -85,B 0,C 180,E1 -8393.644,E2 -8393.644} C_VEL
LIN {X 0,Y 456.592,Z 265.979,A -85,B 0,C 180,E1 -8396.856,E2 -8396.856} C_VEL
LIN {X 0,Y 456.005,Z 261.389,A -85,B 0,C 180,E1 -8397.539,E2 -8397.539} C_VEL
LIN {X 0,Y 453.479,Z 249.163,A -85,B 0,C 180,E1 -8399.459,E2 -8399.459} C_VEL
LIN {X 0,Y 453.466,Z 248.998,A -85,B 0,C 180,E1 -8402.849,E2 -8402.849} C_VEL
LIN {X 0,Y 453.466,Z 249,A -85,B 0,C 180,E1 -8404.989,E2 -8404.989} C_VEL
LIN {X 0,Y 453.432,Z 248.999,A -85,B 0,C 180,E1 -8408.313,E2 -8408.313} C_VEL
LIN {X 0,Y 453.457,Z 248.997,A -85,B 0,C 180,E1 -8410.611,E2 -8410.611} C_VEL
LIN {X 0,Y 453.472,Z 248.995,A -85,B 0,C 180,E1 -8414.527,E2 -8414.527} C_VEL
LIN {X 0,Y 453.426,Z 249,A -85,B 0,C 180,E1 -8418.07,E2 -8418.07} C_VEL
LIN {X 0,Y 453.432,Z 249.002,A -85,B 0,C 180,E1 -8420.801,E2 -8420.801} C_VEL
LIN {X 0,Y 453.432,Z 248.999,A -85,B 0,C 180,E1 -8423.915,E2 -8423.915} C_VEL
LIN {X 0,Y 453.454,Z 249.001,A -85,B 0,C 180,E1 -8426.815,E2 -8426.815} C_VEL
LIN {X 0,Y 453.442,Z 248.998,A -85,B 0,C 180,E1 -8430.266,E2 -8430.266} C_VEL
LIN {X 0,Y 453.411,Z 249.005,A -85,B 0,C 180,E1 -8433.288,E2 -8433.288} C_VEL
LIN {X 0,Y 453.478,Z 248.994,A -85,B 0,C 180,E1 -8436.237,E2 -8436.237} C_VEL
LIN {X 0,Y 453.462,Z 249,A -85,B 0,C 180,E1 -8439.117,E2 -8439.117} C_VEL
LIN {X 0,Y 453.482,Z 248.993,A -85,B 0,C 180,E1 -8441.943,E2 -8441.943} C_VEL
LIN {X 0,Y 453.515,Z 248.996,A -85,B 0,C 180,E1 -8444.726,E2 -8444.726} C_VEL
LIN {X 0,Y 453.542,Z 248.989,A -85,B 0,C 180,E1 -8448.379,E2 -8448.379} C_VEL
LIN {X 0,Y 453.547,Z 248.987,A -85,B 0,C 180,E1 -8451.086,E2 -8451.086} C_VEL
LIN {X 0,Y 453.613,Z 248.977,A -85,B 0,C 180,E1 -8453.774,E2 -8453.774} C_VEL
LIN {X 0,Y 453.698,Z 248.966,A -85,B 0,C 180,E1 -8457.337,E2 -8457.337} C_VEL
LIN {X 0,Y 453.731,Z 248.964,A -85,B 0,C 180,E1 -8460,E2 -8460} C_VEL
LIN {X 0,Y 453.686,Z 248.973,A -85,B 0,C 180,E1 -8462.664,E2 -8462.664} C_VEL
LIN {X 0,Y 453.621,Z 248.981,A -85,B 0,C 180,E1 -8466.226,E2 -8466.226} C_VEL
LIN {X 0,Y 453.541,Z 248.987,A -85,B 0,C 180,E1 -8468.915,E2 -8468.915} C_VEL
LIN {X 0,Y 453.552,Z 248.989,A -85,B 0,C 180,E1 -8472.529,E2 -8472.529} C_VEL
LIN {X 0,Y 453.526,Z 248.995,A -85,B 0,C 180,E1 -8476.197,E2 -8476.197} C_VEL
LIN {X 0,Y 453.506,Z 248.99,A -85,B 0,C 180,E1 -8479.04,E2 -8479.04} C_VEL
LIN {X 0,Y 453.465,Z 248.999,A -85,B 0,C 180,E1 -8481.837,E2 -8481.837} C_VEL
LIN {X 0,Y 453.453,Z 248.997,A -85,B 0,C 180,E1 -8484.738,E2 -8484.738} C_VEL
LIN {X 0,Y 453.451,Z 249.003,A -85,B 0,C 180,E1 -8487.943,E2 -8487.943} C_VEL
LIN {X 0,Y 453.447,Z 248.998,A -85,B 0,C 180,E1 -8490.762,E2 -8490.762} C_VEL
LIN {X 0,Y 453.456,Z 249.004,A -85,B 0,C 180,E1 -8493.915,E2 -8493.915} C_VEL
LIN {X 0,Y 453.425,Z 249.001,A -85,B 0,C 180,E1 -8497.193,E2 -8497.193} C_VEL
LIN {X 0,Y 453.457,Z 248.996,A -85,B 0,C 180,E1 -8500.614,E2 -8500.614} C_VEL
LIN {X 0,Y 453.472,Z 248.994,A -85,B 0,C 180,E1 -8504.529,E2 -8504.529} C_VEL
LIN {X 0,Y 453.425,Z 249.003,A -85,B 0,C 180,E1 -8508.073,E2 -8508.073} C_VEL
LIN {X 0,Y 453.424,Z 249,A -85,B 0,C 180,E1 -8510.805,E2 -8510.805} C_VEL
LIN {X 0,Y 453.435,Z 249.003,A -85,B 0,C 180,E1 -8513.917,E2 -8513.917} C_VEL
LIN {X 0,Y 453.462,Z 248.996,A -85,B 0,C 180,E1 -8516.817,E2 -8516.817} C_VEL
LIN {X 0,Y 453.446,Z 248.998,A -85,B 0,C 180,E1 -8520.267,E2 -8520.267} C_VEL
LIN {X 0,Y 453.422,Z 249.006,A -85,B 0,C 180,E1 -8523.29,E2 -8523.29} C_VEL
LIN {X 0,Y 453.48,Z 248.993,A -85,B 0,C 180,E1 -8526.238,E2 -8526.238} C_VEL
LIN {X 0,Y 453.467,Z 248.999,A -85,B 0,C 180,E1 -8529.118,E2 -8529.118} C_VEL
LIN {X 0,Y 453.471,Z 248.995,A -85,B 0,C 180,E1 -8531.944,E2 -8531.944} C_VEL
LIN {X 0,Y 453.489,Z 248.994,A -85,B 0,C 180,E1 -8534.725,E2 -8534.725} C_VEL
LIN {X 0,Y 453.568,Z 248.989,A -85,B 0,C 180,E1 -8537.472,E2 -8537.472} C_VEL
LIN {X 0,Y 453.568,Z 249.117,A -85,B 0,C 180,E1 -8540.783,E2 -8540.783} C_VEL
LIN {X 0,Y 453.743,Z 250.034,A -85,B 0,C 180,E1 -8540.939,E2 -8540.939} C_VEL
LIN {X 0,Y 457.487,Z 260.604,A -85,B 0,C 180,E1 -8541.26,E2 -8541.26} C_VEL
LIN {X 0,Y 457.573,Z 271.953,A -85,B 0,C 180,E1 -8541.444,E2 -8541.444} C_VEL
LIN {X 0,Y 456.84,Z 277.788,A -85,B 0,C 180,E1 -8541.511,E2 -8541.511} C_VEL
LIN {X 0,Y 451.219,Z 296.767,A -85,B 0,C 180,E1 -8541.618,E2 -8541.618} C_VEL
LIN {X 0,Y 450.437,Z 302.603,A -85,B 0,C 180,E1 -8541.685,E2 -8541.685} C_VEL
LIN {X 0,Y 450.139,Z 338.847,A -85,B 0,C 180,E1 -8542.29,E2 -8542.29} C_VEL
LIN {X 0,Y 450.05,Z 351.616,A -85,B 0,C 180,E1 -8542.683,E2 -8542.683} C_VEL
LIN {X 0,Y 449.781,Z 363.485,A -85,B 0,C 180,E1 -8543.214,E2 -8543.214} C_VEL
LIN {X 0,Y 449.441,Z 375.508,A -85,B 0,C 180,E1 -8543.942,E2 -8543.942} C_VEL
LIN {X 0,Y 448.928,Z 386.893,A -85,B 0,C 180,E1 -8544.836,E2 -8544.836} C_VEL
LIN {X 0,Y 448.416,Z 397.135,A -85,B 0,C 180,E1 -8545.844,E2 -8545.844} C_VEL
LIN {X 0,Y 447.988,Z 405.51,A -85,B 0,C 180,E1 -8546.853,E2 -8546.853} C_VEL
LIN {X 0,Y 447.551,Z 413.242,A -85,B 0,C 180,E1 -8547.976,E2 -8547.976} C_VEL
LIN {X 0,Y 447.057,Z 420.824,A -85,B 0,C 180,E1 -8549.325,E2 -8549.325} C_VEL
LIN {X 0,Y 446.627,Z 427.787,A -85,B 0,C 180,E1 -8550.902,E2 -8550.902} C_VEL
LIN {X 0,Y 446.431,Z 432.422,A -85,B 0,C 180,E1 -8552.256,E2 -8552.256} C_VEL
LIN {X 0,Y 446.191,Z 435.995,A -85,B 0,C 180,E1 -8553.613,E2 -8553.613} C_VEL
LIN {X 0,Y 446.178,Z 437.83,A -85,B 0,C 180,E1 -8554.517,E2 -8554.517} C_VEL
LIN {X 0,Y 446.148,Z 439.218,A -85,B 0,C 180,E1 -8555.424,E2 -8555.424} C_VEL
LIN {X 0,Y 446.087,Z 440.827,A -85,B 0,C 180,E1 -8557.241,E2 -8557.241} C_VEL
LIN {X 0,Y 446.048,Z 441.068,A -85,B 0,C 180,E1 -8558.153,E2 -8558.153} C_VEL
LIN {X 0,Y 446.077,Z 440.297,A -85,B 0,C 180,E1 -8559.98,E2 -8559.98} C_VEL
LIN {X 0,Y 446.128,Z 439.333,A -85,B 0,C 180,E1 -8560.897,E2 -8560.897} C_VEL
LIN {X 0,Y 446.367,Z 436.581,A -85,B 0,C 180,E1 -8562.527,E2 -8562.527} C_VEL
LIN {X 0,Y 446.643,Z 432.518,A -85,B 0,C 180,E1 -8564.117,E2 -8564.117} C_VEL
LIN {X 0,Y 446.965,Z 427.78,A -85,B 0,C 180,E1 -8565.504,E2 -8565.504} C_VEL
LIN {X 0,Y 447.359,Z 421.966,A -85,B 0,C 180,E1 -8566.849,E2 -8566.849} C_VEL
LIN {X 0,Y 447.924,Z 414.173,A -85,B 0,C 180,E1 -8568.289,E2 -8568.289} C_VEL
LIN {X 0,Y 448.512,Z 405.527,A -85,B 0,C 180,E1 -8569.559,E2 -8569.559} C_VEL
LIN {X 0,Y 449.089,Z 395.625,A -85,B 0,C 180,E1 -8570.736,E2 -8570.736} C_VEL
LIN {X 0,Y 449.6,Z 385.909,A -85,B 0,C 180,E1 -8571.672,E2 -8571.672} C_VEL
LIN {X 0,Y 450.117,Z 375.813,A -85,B 0,C 180,E1 -8572.457,E2 -8572.457} C_VEL
LIN {X 0,Y 450.517,Z 364.804,A -85,B 0,C 180,E1 -8573.136,E2 -8573.136} C_VEL
LIN {X 0,Y 450.809,Z 352.583,A -85,B 0,C 180,E1 -8573.698,E2 -8573.698} C_VEL
LIN {X 0,Y 450.929,Z 340.852,A -85,B 0,C 180,E1 -8574.075,E2 -8574.075} C_VEL
LIN {X 0,Y 450.978,Z 317.677,A -85,B 0,C 180,E1 -8574.497,E2 -8574.497} C_VEL
LIN {X 0,Y 451.624,Z 263.249,A -85,B 0,C 180,E1 -8575.371,E2 -8575.371} C_VEL
LIN {X 0,Y 446.662,Z 250.853,A -85,B 0,C 180,E1 -8575.837,E2 -8575.837} C_VEL
LIN {X 0,Y 446.467,Z 249.967,A -85,B 0,C 180,E1 -8576.014,E2 -8576.014} C_VEL
LIN {X 0,Y 446.427,Z 249.877,A -85,B 0,C 180,E1 -8579.211,E2 -8579.211} C_VEL
LIN {X 0,Y 446.418,Z 249.868,A -85,B 0,C 180,E1 -8582.361,E2 -8582.361} C_VEL
LIN {X 0,Y 446.415,Z 249.856,A -85,B 0,C 180,E1 -8585.626,E2 -8585.626} C_VEL
LIN {X 0,Y 446.403,Z 249.88,A -85,B 0,C 180,E1 -8589.031,E2 -8589.031} C_VEL
LIN {X 0,Y 446.384,Z 249.874,A -85,B 0,C 180,E1 -8592.269,E2 -8592.269} C_VEL
LIN {X 0,Y 446.42,Z 249.874,A -85,B 0,C 180,E1 -8595.107,E2 -8595.107} C_VEL
LIN {X 0,Y 446.398,Z 249.88,A -85,B 0,C 180,E1 -8598.605,E2 -8598.605} C_VEL
LIN {X 0,Y 446.395,Z 249.87,A -85,B 0,C 180,E1 -8601.923,E2 -8601.923} C_VEL
LIN {X 0,Y 446.423,Z 249.874,A -85,B 0,C 180,E1 -8605.476,E2 -8605.476} C_VEL
LIN {X 0,Y 446.411,Z 249.861,A -85,B 0,C 180,E1 -8608.699,E2 -8608.699} C_VEL
LIN {X 0,Y 446.42,Z 249.87,A -85,B 0,C 180,E1 -8611.836,E2 -8611.836} C_VEL
LIN {X 0,Y 446.428,Z 249.872,A -85,B 0,C 180,E1 -8614.846,E2 -8614.846} C_VEL
LIN {X 0,Y 446.443,Z 249.85,A -85,B 0,C 180,E1 -8618.245,E2 -8618.245} C_VEL
LIN {X 0,Y 446.444,Z 249.87,A -85,B 0,C 180,E1 -8621.648,E2 -8621.648} C_VEL
LIN {X 0,Y 446.5,Z 249.861,A -85,B 0,C 180,E1 -8624.479,E2 -8624.479} C_VEL
LIN {X 0,Y 446.509,Z 249.865,A -85,B 0,C 180,E1 -8628.193,E2 -8628.193} C_VEL
LIN {X 0,Y 446.518,Z 249.853,A -85,B 0,C 180,E1 -8630.944,E2 -8630.944} C_VEL
LIN {X 0,Y 446.598,Z 249.857,A -85,B 0,C 180,E1 -8633.675,E2 -8633.675} C_VEL
LIN {X 0,Y 446.644,Z 249.842,A -85,B 0,C 180,E1 -8637.294,E2 -8637.294} C_VEL
LIN {X 0,Y 446.709,Z 249.838,A -85,B 0,C 180,E1 -8640,E2 -8640} C_VEL
LIN {X 0,Y 446.655,Z 249.839,A -85,B 0,C 180,E1 -8642.705,E2 -8642.705} C_VEL
LIN {X 0,Y 446.59,Z 249.849,A -85,B 0,C 180,E1 -8646.324,E2 -8646.324} C_VEL
LIN {X 0,Y 446.521,Z 249.859,A -85,B 0,C 180,E1 -8649.056,E2 -8649.056} C_VEL
LIN {X 0,Y 446.515,Z 249.857,A -85,B 0,C 180,E1 -8652.73,E2 -8652.73} C_VEL
LIN {X 0,Y 446.478,Z 249.866,A -85,B 0,C 180,E1 -8656.459,E2 -8656.459} C_VEL
LIN {X 0,Y 446.461,Z 249.873,A -85,B 0,C 180,E1 -8659.303,E2 -8659.303} C_VEL
LIN {X 0,Y 446.409,Z 249.872,A -85,B 0,C 180,E1 -8662.2,E2 -8662.2} C_VEL
LIN {X 0,Y 446.413,Z 249.878,A -85,B 0,C 180,E1 -8665.155,E2 -8665.155} C_VEL
LIN {X 0,Y 446.41,Z 249.865,A -85,B 0,C 180,E1 -8668.184,E2 -8668.184} C_VEL
LIN {X 0,Y 446.387,Z 249.881,A -85,B 0,C 180,E1 -8671.303,E2 -8671.303} C_VEL
LIN {X 0,Y 446.414,Z 249.867,A -85,B 0,C 180,E1 -8674.524,E2 -8674.524} C_VEL
LIN {X 0,Y 446.393,Z 249.875,A -85,B 0,C 180,E1 -8678.077,E2 -8678.077} C_VEL
LIN {X 0,Y 446.395,Z 249.88,A -85,B 0,C 180,E1 -8681.395,E2 -8681.395} C_VEL
LIN {X 0,Y 446.417,Z 249.878,A -85,B 0,C 180,E1 -8685.108,E2 -8685.108} C_VEL
LIN {X 0,Y 446.394,Z 249.882,A -85,B 0,C 180,E1 -8688.606,E2 -8688.606} C_VEL
LIN {X 0,Y 446.39,Z 249.875,A -85,B 0,C 180,E1 -8691.925,E2 -8691.925} C_VEL
LIN {X 0,Y 446.417,Z 249.869,A -85,B 0,C 180,E1 -8695.476,E2 -8695.476} C_VEL
LIN {X 0,Y 446.389,Z 249.877,A -85,B 0,C 180,E1 -8698.698,E2 -8698.698} C_VEL
LIN {X 0,Y 446.434,Z 250.118,A -85,B 0,C 180,E1 -8699.772,E2 -8699.772} C_VEL
LIN {X 0,Y 449.782,Z 265.173,A -85,B 0,C 180,E1 -8702.283,E2 -8702.283} C_VEL
LIN {X 0,Y 450.118,Z 268.965,A -85,B 0,C 180,E1 -8702.871,E2 -8702.871} C_VEL
LIN {X 0,Y 449.015,Z 290.288,A -85,B 0,C 180,E1 -8705.987,E2 -8705.987} C_VEL
LIN {X 0,Y 448.123,Z 310.182,A -85,B 0,C 180,E1 -8708.856,E2 -8708.856} C_VEL
LIN {X 0,Y 447.327,Z 331.763,A -85,B 0,C 180,E1 -8711.921,E2 -8711.921} C_VEL
LIN {X 0,Y 450.005,Z 353.502,A -85,B 0,C 180,E1 -8712.43,E2 -8712.43} C_VEL
LIN {X 0,Y 450.923,Z 363.167,A -85,B 0,C 180,E1 -8712.628,E2 -8712.628} C_VEL
LIN {X 0,Y 450.094,Z 443.152,A -85,B 0,C 180,E1 -8713.938,E2 -8713.938} C_VEL
LIN {X 0,Y 449.54,Z 456.915,A -85,B 0,C 180,E1 -8714.355,E2 -8714.355} C_VEL
LIN {X 0,Y 448.901,Z 469.315,A -85,B 0,C 180,E1 -8714.913,E2 -8714.913} C_VEL
LIN {X 0,Y 448.178,Z 482.031,A -85,B 0,C 180,E1 -8715.701,E2 -8715.701} C_VEL
LIN {X 0,Y 447.464,Z 494.07,A -85,B 0,C 180,E1 -8716.666,E2 -8716.666} C_VEL
LIN {X 0,Y 446.931,Z 504.66,A -85,B 0,C 180,E1 -8717.743,E2 -8717.743} C_VEL
LIN {X 0,Y 446.38,Z 513.782,A -85,B 0,C 180,E1 -8718.88,E2 -8718.88} C_VEL
LIN {X 0,Y 445.944,Z 522.73,A -85,B 0,C 180,E1 -8720.246,E2 -8720.246} C_VEL
LIN {X 0,Y 445.762,Z 529.937,A -85,B 0,C 180,E1 -8721.614,E2 -8721.614} C_VEL
LIN {X 0,Y 445.687,Z 534.853,A -85,B 0,C 180,E1 -8722.753,E2 -8722.753} C_VEL
LIN {X 0,Y 445.654,Z 539.626,A -85,B 0,C 180,E1 -8724.116,E2 -8724.116} C_VEL
LIN {X 0,Y 445.708,Z 543.282,A -85,B 0,C 180,E1 -8725.478,E2 -8725.478} C_VEL
LIN {X 0,Y 445.797,Z 545.159,A -85,B 0,C 180,E1 -8726.384,E2 -8726.384} C_VEL
LIN {X 0,Y 445.744,Z 546.564,A -85,B 0,C 180,E1 -8727.289,E2 -8727.289} C_VEL
LIN {X 0,Y 445.738,Z 548.182,A -85,B 0,C 180,E1 -8729.096,E2 -8729.096} C_VEL
LIN {X 0,Y 445.771,Z 548.373,A -85,B 0,C 180,E1 -8730,E2 -8730} C_VEL
LIN {X 0,Y 445.745,Z 548.127,A -85,B 0,C 180,E1 -8730.903,E2 -8730.903} C_VEL
LIN {X 0,Y 445.751,Z 546.451,A -85,B 0,C 180,E1 -8732.711,E2 -8732.711} C_VEL
LIN {X 0,Y 445.844,Z 544.986,A -85,B 0,C 180,E1 -8733.615,E2 -8733.615} C_VEL
LIN {X 0,Y 445.673,Z 541.91,A -85,B 0,C 180,E1 -8734.975,E2 -8734.975} C_VEL
LIN {X 0,Y 445.726,Z 536.789,A -85,B 0,C 180,E1 -8736.608,E2 -8736.608} C_VEL
LIN {X 0,Y 445.744,Z 530.367,A -85,B 0,C 180,E1 -8738.157,E2 -8738.157} C_VEL
LIN {X 0,Y 445.929,Z 523.189,A -85,B 0,C 180,E1 -8739.525,E2 -8739.525} C_VEL
LIN {X 0,Y 446.279,Z 514.217,A -85,B 0,C 180,E1 -8740.892,E2 -8740.892} C_VEL
LIN {X 0,Y 446.721,Z 505.044,A -85,B 0,C 180,E1 -8742.031,E2 -8742.031} C_VEL
LIN {X 0,Y 447.271,Z 494.392,A -85,B 0,C 180,E1 -8743.106,E2 -8743.106} C_VEL
LIN {X 0,Y 447.758,Z 483.779,A -85,B 0,C 180,E1 -8743.964,E2 -8743.964} C_VEL
LIN {X 0,Y 448.449,Z 471.286,A -85,B 0,C 180,E1 -8744.753,E2 -8744.753} C_VEL
LIN {X 0,Y 449.027,Z 459.447,A -85,B 0,C 180,E1 -8745.314,E2 -8745.314} C_VEL
LIN {X 0,Y 449.515,Z 446.667,A -85,B 0,C 180,E1 -8745.733,E2 -8745.733} C_VEL
LIN {X 0,Y 449.761,Z 428.528,A -85,B 0,C 180,E1 -8746.073,E2 -8746.073} C_VEL
LIN {X 0,Y 450.15,Z 360.757,A -85,B 0,C 180,E1 -8747.155,E2 -8747.155} C_VEL
LIN {X 0,Y 447.141,Z 332.718,A -85,B 0,C 180,E1 -8747.72,E2 -8747.72} C_VEL
LIN {X 0,Y 447.817,Z 311.413,A -85,B 0,C 180,E1 -8750.677,E2 -8750.677} C_VEL
LIN {X 0,Y 448.812,Z 286.314,A -85,B 0,C 180,E1 -8754.232,E2 -8754.232} C_VEL
LIN {X 0,Y 449.639,Z 266.873,A -85,B 0,C 180,E1 -8757.01,E2 -8757.01} C_VEL
LIN {X 0,Y 448.537,Z 260.153,A -85,B 0,C 180,E1 -8758.037,E2 -8758.037} C_VEL
LIN {X 0,Y 446.42,Z 250,A -85,B 0,C 180,E1 -8759.677,E2 -8759.677} C_VEL
LIN {X 0,Y 446.403,Z 249.879,A -85,B 0,C 180,E1 -8762.362,E2 -8762.362} C_VEL
LIN {X 0,Y 446.415,Z 249.879,A -85,B 0,C 180,E1 -8765.05,E2 -8765.05} C_VEL
LIN {X 0,Y 446.386,Z 249.877,A -85,B 0,C 180,E1 -8768.074,E2 -8768.074} C_VEL
LIN {X 0,Y 446.389,Z 249.883,A -85,B 0,C 180,E1 -8771.394,E2 -8771.394} C_VEL
LIN {X 0,Y 446.441,Z 249.876,A -85,B 0,C 180,E1 -8775.103,E2 -8775.103} C_VEL
LIN {X 0,Y 446.391,Z 249.878,A -85,B 0,C 180,E1 -8778.605,E2 -8778.605} C_VEL
LIN {X 0,Y 446.39,Z 249.877,A -85,B 0,C 180,E1 -8781.923,E2 -8781.923} C_VEL
LIN {X 0,Y 446.403,Z 249.878,A -85,B 0,C 180,E1 -8785.475,E2 -8785.475} C_VEL
LIN {X 0,Y 446.379,Z 249.881,A -85,B 0,C 180,E1 -8788.697,E2 -8788.697} C_VEL
LIN {X 0,Y 446.394,Z 249.876,A -85,B 0,C 180,E1 -8791.84,E2 -8791.84} C_VEL
LIN {X 0,Y 446.4,Z 249.882,A -85,B 0,C 180,E1 -8794.844,E2 -8794.844} C_VEL
LIN {X 0,Y 446.435,Z 249.872,A -85,B 0,C 180,E1 -8798.245,E2 -8798.245} C_VEL
LIN {X 0,Y 446.434,Z 249.871,A -85,B 0,C 180,E1 -8801.648,E2 -8801.648} C_VEL
LIN {X 0,Y 446.462,Z 249.871,A -85,B 0,C 180,E1 -8804.478,E2 -8804.478} C_VEL
LIN {X 0,Y 446.502,Z 249.864,A -85,B 0,C 180,E1 -8808.193,E2 -8808.193} C_VEL
LIN {X 0,Y 446.498,Z 249.867,A -85,B 0,C 180,E1 -8810.944,E2 -8810.944} C_VEL
LIN {X 0,Y 446.584,Z 249.852,A -85,B 0,C 180,E1 -8813.676,E2 -8813.676} C_VEL
LIN {X 0,Y 446.648,Z 249.845,A -85,B 0,C 180,E1 -8817.295,E2 -8817.295} C_VEL
LIN {X 0,Y 446.682,Z 249.842,A -85,B 0,C 180,E1 -8820,E2 -8820} C_VEL
LIN {X 0,Y 446.636,Z 249.85,A -85,B 0,C 180,E1 -8822.706,E2 -8822.706} C_VEL
LIN {X 0,Y 446.591,Z 249.858,A -85,B 0,C 180,E1 -8826.325,E2 -8826.325} C_VEL
LIN {X 0,Y 446.492,Z 249.864,A -85,B 0,C 180,E1 -8829.057,E2 -8829.057} C_VEL
LIN {X 0,Y 446.51,Z 249.864,A -85,B 0,C 180,E1 -8832.73,E2 -8832.73} C_VEL
LIN {X 0,Y 446.473,Z 249.871,A -85,B 0,C 180,E1 -8836.46,E2 -8836.46} C_VEL
LIN {X 0,Y 446.457,Z 249.868,A -85,B 0,C 180,E1 -8839.304,E2 -8839.304} C_VEL
LIN {X 0,Y 446.406,Z 249.882,A -85,B 0,C 180,E1 -8842.201,E2 -8842.201} C_VEL
LIN {X 0,Y 446.404,Z 249.875,A -85,B 0,C 180,E1 -8845.156,E2 -8845.156} C_VEL
LIN {X 0,Y 446.407,Z 249.88,A -85,B 0,C 180,E1 -8848.184,E2 -8848.184} C_VEL
LIN {X 0,Y 446.398,Z 249.876,A -85,B 0,C 180,E1 -8851.302,E2 -8851.302} C_VEL
LIN {X 0,Y 446.41,Z 249.875,A -85,B 0,C 180,E1 -8854.525,E2 -8854.525} C_VEL
LIN {X 0,Y 446.386,Z 249.882,A -85,B 0,C 180,E1 -8858.077,E2 -8858.077} C_VEL
LIN {X 0,Y 446.388,Z 249.879,A -85,B 0,C 180,E1 -8861.396,E2 -8861.396} C_VEL
LIN {X 0,Y 446.412,Z 249.874,A -85,B 0,C 180,E1 -8864.893,E2 -8864.893} C_VEL
LIN {X 0,Y 446.391,Z 249.876,A -85,B 0,C 180,E1 -8868.606,E2 -8868.606} C_VEL
LIN {X 0,Y 446.39,Z 249.881,A -85,B 0,C 180,E1 -8871.926,E2 -8871.926} C_VEL
LIN {X 0,Y 446.409,Z 249.88,A -85,B 0,C 180,E1 -8875.477,E2 -8875.477} C_VEL
LIN {X 0,Y 446.386,Z 249.877,A -85,B 0,C 180,E1 -8878.699,E2 -8878.699} C_VEL
LIN {X 0,Y 446.4,Z 249.878,A -85,B 0,C 180,E1 -8881.843,E2 -8881.843} C_VEL
LIN {X 0,Y 446.412,Z 249.875,A -85,B 0,C 180,E1 -8884.846,E2 -8884.846} C_VEL
LIN {X 0,Y 446.446,Z 249.869,A -85,B 0,C 180,E1 -8888.247,E2 -8888.247} C_VEL
LIN {X 0,Y 446.419,Z 249.876,A -85,B 0,C 180,E1 -8891.648,E2 -8891.648} C_VEL
LIN {X 0,Y 446.433,Z 249.871,A -85,B 0,C 180,E1 -8894.478,E2 -8894.478} C_VEL
LIN {X 0,Y 446.519,Z 249.868,A -85,B 0,C 180,E1 -8897.385,E2 -8897.385} C_VEL
LIN {X 0,Y 446.544,Z 250.003,A -85,B 0,C 180,E1 -8900.54,E2 -8900.54} C_VEL
LIN {X 0,Y 446.756,Z 250.985,A -85,B 0,C 180,E1 -8900.698,E2 -8900.698} C_VEL
LIN {X 0,Y 450.771,Z 262.322,A -85,B 0,C 180,E1 -8901.045,E2 -8901.045} C_VEL
LIN {X 0,Y 450.437,Z 302.603,A -85,B 0,C 180,E1 -8901.685,E2 -8901.685} C_VEL
LIN {X 0,Y 449.615,Z 308.449,A -85,B 0,C 180,E1 -8901.751,E2 -8901.751} C_VEL
LIN {X 0,Y 443.897,Z 327.426,A -85,B 0,C 180,E1 -8901.862,E2 -8901.862} C_VEL
LIN {X 0,Y 443.353,Z 333.258,A -85,B 0,C 180,E1 -8901.941,E2 -8901.941} C_VEL
LIN {X 0,Y 443.227,Z 346.279,A -85,B 0,C 180,E1 -8902.255,E2 -8902.255} C_VEL
LIN {X 0,Y 443.011,Z 359.472,A -85,B 0,C 180,E1 -8902.767,E2 -8902.767} C_VEL
LIN {X 0,Y 442.747,Z 370.963,A -85,B 0,C 180,E1 -8903.392,E2 -8903.392} C_VEL
LIN {X 0,Y 442.303,Z 382.166,A -85,B 0,C 180,E1 -8904.187,E2 -8904.187} C_VEL
LIN {X 0,Y 441.744,Z 393.531,A -85,B 0,C 180,E1 -8905.209,E2 -8905.209} C_VEL
LIN {X 0,Y 441.214,Z 403.607,A -85,B 0,C 180,E1 -8906.347,E2 -8906.347} C_VEL
LIN {X 0,Y 440.687,Z 411.806,A -85,B 0,C 180,E1 -8907.487,E2 -8907.487} C_VEL
LIN {X 0,Y 440.233,Z 419.814,A -85,B 0,C 180,E1 -8908.857,E2 -8908.857} C_VEL
LIN {X 0,Y 439.864,Z 425.292,A -85,B 0,C 180,E1 -8910,E2 -8910} C_VEL
LIN {X 0,Y 439.529,Z 430.642,A -85,B 0,C 180,E1 -8911.375,E2 -8911.375} C_VEL
LIN {X 0,Y 439.29,Z 434.837,A -85,B 0,C 180,E1 -8912.751,E2 -8912.751} C_VEL
LIN {X 0,Y 439.146,Z 437.068,A -85,B 0,C 180,E1 -8913.671,E2 -8913.671} C_VEL
LIN {X 0,Y 439.143,Z 438.844,A -85,B 0,C 180,E1 -8914.59,E2 -8914.59} C_VEL
LIN {X 0,Y 439.106,Z 440.185,A -85,B 0,C 180,E1 -8915.511,E2 -8915.511} C_VEL
LIN {X 0,Y 439.051,Z 441.728,A -85,B 0,C 180,E1 -8917.358,E2 -8917.358} C_VEL
LIN {X 0,Y 439.004,Z 441.91,A -85,B 0,C 180,E1 -8918.284,E2 -8918.284} C_VEL
LIN {X 0,Y 439.06,Z 441.063,A -85,B 0,C 180,E1 -8920.141,E2 -8920.141} C_VEL
LIN {X 0,Y 439.113,Z 440.066,A -85,B 0,C 180,E1 -8921.073,E2 -8921.073} C_VEL
LIN {X 0,Y 439.366,Z 437.401,A -85,B 0,C 180,E1 -8922.643,E2 -8922.643} C_VEL
LIN {X 0,Y 439.689,Z 433.067,A -85,B 0,C 180,E1 -8924.345,E2 -8924.345} C_VEL
LIN {X 0,Y 440.033,Z 428.249,A -85,B 0,C 180,E1 -8925.755,E2 -8925.755} C_VEL
LIN {X 0,Y 440.467,Z 422.345,A -85,B 0,C 180,E1 -8927.121,E2 -8927.121} C_VEL
LIN {X 0,Y 440.984,Z 415.807,A -85,B 0,C 180,E1 -8928.346,E2 -8928.346} C_VEL
LIN {X 0,Y 441.618,Z 407.1,A -85,B 0,C 180,E1 -8929.676,E2 -8929.676} C_VEL
LIN {X 0,Y 442.18,Z 397.722,A -85,B 0,C 180,E1 -8930.832,E2 -8930.832} C_VEL
LIN {X 0,Y 442.805,Z 386.965,A -85,B 0,C 180,E1 -8931.899,E2 -8931.899} C_VEL
LIN {X 0,Y 443.311,Z 377.268,A -85,B 0,C 180,E1 -8932.671,E2 -8932.671} C_VEL
LIN {X 0,Y 443.792,Z 366.004,A -85,B 0,C 180,E1 -8933.384,E2 -8933.384} C_VEL
LIN {X 0,Y 444.11,Z 353.929,A -85,B 0,C 180,E1 -8933.954,E2 -8933.954} C_VEL
LIN {X 0,Y 444.239,Z 342.425,A -85,B 0,C 180,E1 -8934.337,E2 -8934.337} C_VEL
LIN {X 0,Y 444.257,Z 323.388,A -85,B 0,C 180,E1 -8934.706,E2 -8934.706} C_VEL
LIN {X 0,Y 444.912,Z 264.829,A -85,B 0,C 180,E1 -8935.665,E2 -8935.665} C_VEL
LIN {X 0,Y 439.599,Z 251.683,A -85,B 0,C 180,E1 -8936.178,E2 -8936.178} C_VEL
LIN {X 0,Y 439.416,Z 250.811,A -85,B 0,C 180,E1 -8936.378,E2 -8936.378} C_VEL
LIN {X 0,Y 439.374,Z 250.749,A -85,B 0,C 180,E1 -8939.726,E2 -8939.726} C_VEL
LIN {X 0,Y 439.372,Z 250.754,A -85,B 0,C 180,E1 -8942.946,E2 -8942.946} C_VEL
LIN {X 0,Y 439.37,Z 250.726,A -85,B 0,C 180,E1 -8946.287,E2 -8946.287} C_VEL
LIN {X 0,Y 439.359,Z 250.756,A -85,B 0,C 180,E1 -8949.779,E2 -8949.779} C_VEL
LIN {X 0,Y 439.335,Z 250.754,A -85,B 0,C 180,E1 -8952.62,E2 -8952.62} C_VEL
LIN {X 0,Y 439.374,Z 250.751,A -85,B 0,C 180,E1 -8955.267,E2 -8955.267} C_VEL
LIN {X 0,Y 439.361,Z 250.758,A -85,B 0,C 180,E1 -8958.747,E2 -8958.747} C_VEL
LIN {X 0,Y 439.353,Z 250.748,A -85,B 0,C 180,E1 -8961.61,E2 -8961.61} C_VEL
LIN {X 0,Y 439.391,Z 250.752,A -85,B 0,C 180,E1 -8964.843,E2 -8964.843} C_VEL
LIN {X 0,Y 439.368,Z 250.745,A -85,B 0,C 180,E1 -8968.139,E2 -8968.139} C_VEL
LIN {X 0,Y 439.396,Z 250.743,A -85,B 0,C 180,E1 -8971.606,E2 -8971.606} C_VEL
LIN {X 0,Y 439.368,Z 250.755,A -85,B 0,C 180,E1 -8974.412,E2 -8974.412} C_VEL
LIN {X 0,Y 439.358,Z 250.736,A -85,B 0,C 180,E1 -8977.424,E2 -8977.424} C_VEL
LIN {X 0,Y 439.435,Z 250.74,A -85,B 0,C 180,E1 -8980.663,E2 -8980.663} C_VEL
LIN {X 0,Y 439.455,Z 250.74,A -85,B 0,C 180,E1 -8984.224,E2 -8984.224} C_VEL
LIN {X 0,Y 439.476,Z 250.744,A -85,B 0,C 180,E1 -8988.001,E2 -8988.001} C_VEL
LIN {X 0,Y 439.495,Z 250.735,A -85,B 0,C 180,E1 -8991.725,E2 -8991.725} C_VEL
LIN {X 0,Y 439.589,Z 250.723,A -85,B 0,C 180,E1 -8994.495,E2 -8994.495} C_VEL
LIN {X 0,Y 439.617,Z 250.723,A -85,B 0,C 180,E1 -8998.168,E2 -8998.168} C_VEL
LIN {X 0,Y 439.66,Z 250.716,A -85,B 0,C 180,E1 -9000,E2 -9000} C_VEL
LIN {X 0,Y 439.607,Z 250.717,A -85,B 0,C 180,E1 -9002.749,E2 -9002.749} C_VEL
LIN {X 0,Y 439.542,Z 250.726,A -85,B 0,C 180,E1 -9006.426,E2 -9006.426} C_VEL
LIN {X 0,Y 439.485,Z 250.737,A -85,B 0,C 180,E1 -9009.202,E2 -9009.202} C_VEL
LIN {X 0,Y 439.458,Z 250.738,A -85,B 0,C 180,E1 -9012.938,E2 -9012.938} C_VEL
LIN {X 0,Y 439.438,Z 250.743,A -85,B 0,C 180,E1 -9016.347,E2 -9016.347} C_VEL
LIN {X 0,Y 439.395,Z 250.753,A -85,B 0,C 180,E1 -9019.627,E2 -9019.627} C_VEL
LIN {X 0,Y 439.355,Z 250.751,A -85,B 0,C 180,E1 -9022.576,E2 -9022.576} C_VEL
LIN {X 0,Y 439.358,Z 250.751,A -85,B 0,C 180,E1 -9025.588,E2 -9025.588} C_VEL
LIN {X 0,Y 439.374,Z 250.743,A -85,B 0,C 180,E1 -9028.677,E2 -9028.677} C_VEL
LIN {X 0,Y 439.348,Z 250.753,A -85,B 0,C 180,E1 -9032.027,E2 -9032.027} C_VEL
LIN {X 0,Y 439.381,Z 250.754,A -85,B 0,C 180,E1 -9035.339,E2 -9035.339} C_VEL
LIN {X 0,Y 439.35,Z 250.752,A -85,B 0,C 180,E1 -9038.598,E2 -9038.598} C_VEL
LIN {X 0,Y 439.358,Z 250.758,A -85,B 0,C 180,E1 -9041.253,E2 -9041.253} C_VEL
LIN {X 0,Y 439.392,Z 250.754,A -85,B 0,C 180,E1 -9044.73,E2 -9044.73} C_VEL
LIN {X 0,Y 439.342,Z 250.757,A -85,B 0,C 180,E1 -9047.79,E2 -9047.79} C_VEL
LIN {X 0,Y 439.356,Z 250.744,A -85,B 0,C 180,E1 -9050.22,E2 -9050.22} C_VEL
LIN {X 0,Y 439.361,Z 250.756,A -85,B 0,C 180,E1 -9053.712,E2 -9053.712} C_VEL
LIN {X 0,Y 439.365,Z 250.754,A -85,B 0,C 180,E1 -9057.054,E2 -9057.054} C_VEL
LIN {X 0,Y 439.41,Z 250.893,A -85,B 0,C 180,E1 -9059.445,E2 -9059.445} C_VEL
LIN {X 0,Y 442.827,Z 266.329,A -85,B 0,C 180,E1 -9062.084,E2 -9062.084} C_VEL
LIN {X 0,Y 443.233,Z 270.557,A -85,B 0,C 180,E1 -9062.753,E2 -9062.753} C_VEL
LIN {X 0,Y 442.184,Z 289.657,A -85,B 0,C 180,E1 -9065.592,E2 -9065.592} C_VEL
LIN {X 0,Y 441.264,Z 309.546,A -85,B 0,C 180,E1 -9068.511,E2 -9068.511} C_VEL
LIN {X 0,Y 440.379,Z 330.852,A -85,B 0,C 180,E1 -9071.587,E2 -9071.587} C_VEL
LIN {X 0,Y 443.336,Z 354.788,A -85,B 0,C 180,E1 -9072.156,E2 -9072.156} C_VEL
LIN {X 0,Y 444.185,Z 364.341,A -85,B 0,C 180,E1 -9072.356,E2 -9072.356} C_VEL
LIN {X 0,Y 443.386,Z 441.227,A -85,B 0,C 180,E1 -9073.63,E2 -9073.63} C_VEL
LIN {X 0,Y 442.836,Z 454.578,A -85,B 0,C 180,E1 -9074.023,E2 -9074.023} C_VEL
LIN {X 0,Y 442.075,Z 467.937,A -85,B 0,C 180,E1 -9074.616,E2 -9074.616} C_VEL
LIN {X 0,Y 441.386,Z 479.987,A -85,B 0,C 180,E1 -9075.358,E2 -9075.358} C_VEL
LIN {X 0,Y 440.624,Z 491.494,A -85,B 0,C 180,E1 -9076.271,E2 -9076.271} C_VEL
LIN {X 0,Y 440.158,Z 500.935,A -85,B 0,C 180,E1 -9077.2,E2 -9077.2} C_VEL
LIN {X 0,Y 439.507,Z 509.693,A -85,B 0,C 180,E1 -9078.236,E2 -9078.236} C_VEL
LIN {X 0,Y 439.111,Z 517.808,A -85,B 0,C 180,E1 -9079.394,E2 -9079.394} C_VEL
LIN {X 0,Y 438.783,Z 525.805,A -85,B 0,C 180,E1 -9080.783,E2 -9080.783} C_VEL
LIN {X 0,Y 438.645,Z 532.233,A -85,B 0,C 180,E1 -9082.173,E2 -9082.173} C_VEL
LIN {X 0,Y 438.594,Z 537.376,A -85,B 0,C 180,E1 -9083.559,E2 -9083.559} C_VEL
LIN {X 0,Y 438.562,Z 541.371,A -85,B 0,C 180,E1 -9084.943,E2 -9084.943} C_VEL
LIN {X 0,Y 438.719,Z 544.342,A -85,B 0,C 180,E1 -9086.326,E2 -9086.326} C_VEL
LIN {X 0,Y 438.691,Z 545.742,A -85,B 0,C 180,E1 -9087.245,E2 -9087.245} C_VEL
LIN {X 0,Y 438.685,Z 547.344,A -85,B 0,C 180,E1 -9089.082,E2 -9089.082} C_VEL
LIN {X 0,Y 438.723,Z 547.519,A -85,B 0,C 180,E1 -9090,E2 -9090} C_VEL
LIN {X 0,Y 438.695,Z 547.265,A -85,B 0,C 180,E1 -9090.918,E2 -9090.918} C_VEL
LIN {X 0,Y 438.699,Z 545.571,A -85,B 0,C 180,E1 -9092.754,E2 -9092.754} C_VEL
LIN {X 0,Y 438.798,Z 544.088,A -85,B 0,C 180,E1 -9093.673,E2 -9093.673} C_VEL
LIN {X 0,Y 438.599,Z 540.989,A -85,B 0,C 180,E1 -9095.056,E2 -9095.056} C_VEL
LIN {X 0,Y 438.644,Z 536.255,A -85,B 0,C 180,E1 -9096.6,E2 -9096.6} C_VEL
LIN {X 0,Y 438.663,Z 529.392,A -85,B 0,C 180,E1 -9098.29,E2 -9098.29} C_VEL
LIN {X 0,Y 438.868,Z 522.171,A -85,B 0,C 180,E1 -9099.679,E2 -9099.679} C_VEL
LIN {X 0,Y 439.256,Z 513.164,A -85,B 0,C 180,E1 -9101.069,E2 -9101.069} C_VEL
LIN {X 0,Y 439.772,Z 503.955,A -85,B 0,C 180,E1 -9102.224,E2 -9102.224} C_VEL
LIN {X 0,Y 440.214,Z 494.417,A -85,B 0,C 180,E1 -9103.208,E2 -9103.208} C_VEL
LIN {X 0,Y 440.728,Z 484.118,A -85,B 0,C 180,E1 -9104.074,E2 -9104.074} C_VEL
LIN {X 0,Y 441.442,Z 471.931,A -85,B 0,C 180,E1 -9104.875,E2 -9104.875} C_VEL
LIN {X 0,Y 442.088,Z 459.232,A -85,B 0,C 180,E1 -9105.501,E2 -9105.501} C_VEL
LIN {X 0,Y 442.6,Z 446.908,A -85,B 0,C 180,E1 -9105.926,E2 -9105.926} C_VEL
LIN {X 0,Y 442.813,Z 432.993,A -85,B 0,C 180,E1 -9106.214,E2 -9106.214} C_VEL
LIN {X 0,Y 443.31,Z 361.601,A -85,B 0,C 180,E1 -9107.366,E2 -9107.366} C_VEL
LIN {X 0,Y 440.115,Z 331.674,A -85,B 0,C 180,E1 -9107.992,E2 -9107.992} C_VEL
LIN {X 0,Y 440.796,Z 311.987,A -85,B 0,C 180,E1 -9110.777,E2 -9110.777} C_VEL
LIN {X 0,Y 441.846,Z 286.622,A -85,B 0,C 180,E1 -9114.427,E2 -9114.427} C_VEL
LIN {X 0,Y 442.674,Z 267.259,A -85,B 0,C 180,E1 -9117.243,E2 -9117.243} C_VEL
LIN {X 0,Y 439.385,Z 250.928,A -85,B 0,C 180,E1 -9119.861,E2 -9119.861} C_VEL
LIN {X 0,Y 439.362,Z 250.756,A -85,B 0,C 180,E1 -9122.946,E2 -9122.946} C_VEL
LIN {X 0,Y 439.358,Z 250.752,A -85,B 0,C 180,E1 -9126.287,E2 -9126.287} C_VEL
LIN {X 0,Y 439.341,Z 250.755,A -85,B 0,C 180,E1 -9128.598,E2 -9128.598} C_VEL
LIN {X 0,Y 439.338,Z 250.755,A -85,B 0,C 180,E1 -9132.209,E2 -9132.209} C_VEL
LIN {X 0,Y 439.388,Z 250.756,A -85,B 0,C 180,E1 -9135.269,E2 -9135.269} C_VEL
LIN {X 0,Y 439.344,Z 250.76,A -85,B 0,C 180,E1 -9139.015,E2 -9139.015} C_VEL
LIN {X 0,Y 439.348,Z 250.756,A -85,B 0,C 180,E1 -9141.61,E2 -9141.61} C_VEL
LIN {X 0,Y 439.379,Z 250.754,A -85,B 0,C 180,E1 -9144.842,E2 -9144.842} C_VEL
LIN {X 0,Y 439.334,Z 250.755,A -85,B 0,C 180,E1 -9148.136,E2 -9148.136} C_VEL
LIN {X 0,Y 439.368,Z 250.754,A -85,B 0,C 180,E1 -9151.323,E2 -9151.323} C_VEL
LIN {X 0,Y 439.341,Z 250.756,A -85,B 0,C 180,E1 -9154.411,E2 -9154.411} C_VEL
LIN {X 0,Y 439.349,Z 250.755,A -85,B 0,C 180,E1 -9157.424,E2 -9157.424} C_VEL
LIN {X 0,Y 439.428,Z 250.749,A -85,B 0,C 180,E1 -9160.663,E2 -9160.663} C_VEL
LIN {X 0,Y 439.431,Z 250.745,A -85,B 0,C 180,E1 -9164.223,E2 -9164.223} C_VEL
LIN {X 0,Y 439.469,Z 250.739,A -85,B 0,C 180,E1 -9168.001,E2 -9168.001} C_VEL
LIN {X 0,Y 439.467,Z 250.739,A -85,B 0,C 180,E1 -9171.725,E2 -9171.725} C_VEL
LIN {X 0,Y 439.576,Z 250.732,A -85,B 0,C 180,E1 -9174.495,E2 -9174.495} C_VEL
LIN {X 0,Y 439.616,Z 250.723,A -85,B 0,C 180,E1 -9178.168,E2 -9178.168} C_VEL
LIN {X 0,Y 439.57,Z 250.728,A -85,B 0,C 180,E1 -9180.916,E2 -9180.916} C_VEL
LIN {X 0,Y 439.587,Z 250.728,A -85,B 0,C 180,E1 -9182.749,E2 -9182.749} C_VEL
LIN {X 0,Y 439.544,Z 250.737,A -85,B 0,C 180,E1 -9186.427,E2 -9186.427} C_VEL
LIN {X 0,Y 439.458,Z 250.74,A -85,B 0,C 180,E1 -9189.203,E2 -9189.203} C_VEL
LIN {X 0,Y 439.453,Z 250.741,A -85,B 0,C 180,E1 -9192.938,E2 -9192.938} C_VEL
LIN {X 0,Y 439.433,Z 250.749,A -85,B 0,C 180,E1 -9196.348,E2 -9196.348} C_VEL
LIN {X 0,Y 439.39,Z 250.75,A -85,B 0,C 180,E1 -9199.627,E2 -9199.627} C_VEL
LIN {X 0,Y 439.351,Z 250.756,A -85,B 0,C 180,E1 -9202.577,E2 -9202.577} C_VEL
LIN {X 0,Y 439.352,Z 250.755,A -85,B 0,C 180,E1 -9205.589,E2 -9205.589} C_VEL
LIN {X 0,Y 439.372,Z 250.752,A -85,B 0,C 180,E1 -9208.677,E2 -9208.677} C_VEL
LIN {X 0,Y 439.353,Z 250.76,A -85,B 0,C 180,E1 -9212.03,E2 -9212.03} C_VEL
LIN {X 0,Y 439.378,Z 250.751,A -85,B 0,C 180,E1 -9215.34,E2 -9215.34} C_VEL
LIN {X 0,Y 439.342,Z 250.755,A -85,B 0,C 180,E1 -9218.6,E2 -9218.6} C_VEL
LIN {X 0,Y 439.351,Z 250.755,A -85,B 0,C 180,E1 -9221.253,E2 -9221.253} C_VEL
LIN {X 0,Y 439.366,Z 250.751,A -85,B 0,C 180,E1 -9224.734,E2 -9224.734} C_VEL
LIN {X 0,Y 439.339,Z 250.762,A -85,B 0,C 180,E1 -9227.791,E2 -9227.791} C_VEL
LIN {X 0,Y 439.355,Z 250.754,A -85,B 0,C 180,E1 -9230.221,E2 -9230.221} C_VEL
LIN {X 0,Y 439.36,Z 250.759,A -85,B 0,C 180,E1 -9233.713,E2 -9233.713} C_VEL
LIN {X 0,Y 439.339,Z 250.757,A -85,B 0,C 180,E1 -9237.052,E2 -9237.052} C_VEL
LIN {X 0,Y 439.355,Z 250.753,A -85,B 0,C 180,E1 -9240.273,E2 -9240.273} C_VEL
LIN {X 0,Y 439.354,Z 250.76,A -85,B 0,C 180,E1 -9243.392,E2 -9243.392} C_VEL
LIN {X 0,Y 439.356,Z 250.753,A -85,B 0,C 180,E1 -9246.429,E2 -9246.429} C_VEL
LIN {X 0,Y 439.369,Z 250.758,A -85,B 0,C 180,E1 -9249.397,E2 -9249.397} C_VEL
LIN {X 0,Y 439.383,Z 250.749,A -85,B 0,C 180,E1 -9252.308,E2 -9252.308} C_VEL
LIN {X 0,Y 439.379,Z 250.756,A -85,B 0,C 180,E1 -9255.172,E2 -9255.172} C_VEL
LIN {X 0,Y 439.479,Z 250.74,A -85,B 0,C 180,E1 -9258.002,E2 -9258.002} C_VEL
LIN {X 0,Y 439.485,Z 250.871,A -85,B 0,C 180,E1 -9260.276,E2 -9260.276} C_VEL
LIN {X 0,Y 439.694,Z 251.859,A -85,B 0,C 180,E1 -9260.443,E2 -9260.443} C_VEL
LIN {X 0,Y 443.913,Z 263.709,A -85,B 0,C 180,E1 -9260.813,E2 -9260.813} C_VEL
LIN {X 0,Y 443.353,Z 333.258,A -85,B 0,C 180,E1 -9261.941,E2 -9261.941} C_VEL
LIN {X 0,Y 442.735,Z 339.113,A -85,B 0,C 180,E1 -9262.035,E2 -9262.035} C_VEL
LIN {X 0,Y 439.702,Z 348.542,A -85,B 0,C 180,E1 -9262.193,E2 -9262.193} C_VEL
LIN {X 0,Y 436.689,Z 357.772,A -85,B 0,C 180,E1 -9262.453,E2 -9262.453} C_VEL
LIN {X 0,Y 436.094,Z 363.3,A -85,B 0,C 180,E1 -9262.705,E2 -9262.705} C_VEL
LIN {X 0,Y 435.758,Z 374.989,A -85,B 0,C 180,E1 -9263.402,E2 -9263.402} C_VEL
LIN {X 0,Y 435.289,Z 385.577,A -85,B 0,C 180,E1 -9264.209,E2 -9264.209} C_VEL
LIN {X 0,Y 434.751,Z 396.391,A -85,B 0,C 180,E1 -9265.248,E2 -9265.248} C_VEL
LIN {X 0,Y 434.108,Z 406.931,A -85,B 0,C 180,E1 -9266.52,E2 -9266.52} C_VEL
LIN {X 0,Y 433.623,Z 414.712,A -85,B 0,C 180,E1 -9267.678,E2 -9267.678} C_VEL
LIN {X 0,Y 433.094,Z 422.349,A -85,B 0,C 180,E1 -9269.071,E2 -9269.071} C_VEL
LIN {X 0,Y 432.691,Z 428.457,A -85,B 0,C 180,E1 -9270.466,E2 -9270.466} C_VEL
LIN {X 0,Y 432.458,Z 433.308,A -85,B 0,C 180,E1 -9271.863,E2 -9271.863} C_VEL
LIN {X 0,Y 432.179,Z 437.085,A -85,B 0,C 180,E1 -9273.263,E2 -9273.263} C_VEL
LIN {X 0,Y 432.11,Z 439.841,A -85,B 0,C 180,E1 -9274.665,E2 -9274.665} C_VEL
LIN {X 0,Y 432.066,Z 441.15,A -85,B 0,C 180,E1 -9275.601,E2 -9275.601} C_VEL
LIN {X 0,Y 432.001,Z 442.623,A -85,B 0,C 180,E1 -9277.478,E2 -9277.478} C_VEL
LIN {X 0,Y 431.987,Z 442.479,A -85,B 0,C 180,E1 -9279.363,E2 -9279.363} C_VEL
LIN {X 0,Y 432.052,Z 441.831,A -85,B 0,C 180,E1 -9280.308,E2 -9280.308} C_VEL
LIN {X 0,Y 432.102,Z 440.789,A -85,B 0,C 180,E1 -9281.255,E2 -9281.255} C_VEL
LIN {X 0,Y 432.352,Z 438.246,A -85,B 0,C 180,E1 -9282.754,E2 -9282.754} C_VEL
LIN {X 0,Y 432.629,Z 435.018,A -85,B 0,C 180,E1 -9284.103,E2 -9284.103} C_VEL
LIN {X 0,Y 432.981,Z 430.516,A -85,B 0,C 180,E1 -9285.535,E2 -9285.535} C_VEL
LIN {X 0,Y 433.517,Z 423.621,A -85,B 0,C 180,E1 -9287.209,E2 -9287.209} C_VEL
LIN {X 0,Y 434.157,Z 416.093,A -85,B 0,C 180,E1 -9288.645,E2 -9288.645} C_VEL
LIN {X 0,Y 434.736,Z 408.329,A -85,B 0,C 180,E1 -9289.846,E2 -9289.846} C_VEL
LIN {X 0,Y 435.372,Z 398.755,A -85,B 0,C 180,E1 -9291.049,E2 -9291.049} C_VEL
LIN {X 0,Y 436.041,Z 388.04,A -85,B 0,C 180,E1 -9292.133,E2 -9292.133} C_VEL
LIN {X 0,Y 436.651,Z 377.223,A -85,B 0,C 180,E1 -9293.002,E2 -9293.002} C_VEL
LIN {X 0,Y 437.12,Z 366.111,A -85,B 0,C 180,E1 -9293.7,E2 -9293.7} C_VEL
LIN {X 0,Y 437.423,Z 353.753,A -85,B 0,C 180,E1 -9294.281,E2 -9294.281} C_VEL
LIN {X 0,Y 437.547,Z 342.412,A -85,B 0,C 180,E1 -9294.653,E2 -9294.653} C_VEL
LIN {X 0,Y 437.614,Z 318.569,A -85,B 0,C 180,E1 -9295.099,E2 -9295.099} C_VEL
LIN {X 0,Y 438.25,Z 266.474,A -85,B 0,C 180,E1 -9295.966,E2 -9295.966} C_VEL
LIN {X 0,Y 432.547,Z 252.59,A -85,B 0,C 180,E1 -9296.525,E2 -9296.525} C_VEL
LIN {X 0,Y 432.345,Z 251.698,A -85,B 0,C 180,E1 -9296.726,E2 -9296.726} C_VEL
LIN {X 0,Y 432.33,Z 251.633,A -85,B 0,C 180,E1 -9299.188,E2 -9299.188} C_VEL
LIN {X 0,Y 432.323,Z 251.624,A -85,B 0,C 180,E1 -9302.443,E2 -9302.443} C_VEL
LIN {X 0,Y 432.336,Z 251.604,A -85,B 0,C 180,E1 -9305.817,E2 -9305.817} C_VEL
LIN {X 0,Y 432.301,Z 251.636,A -85,B 0,C 180,E1 -9309.348,E2 -9309.348} C_VEL
LIN {X 0,Y 432.304,Z 251.627,A -85,B 0,C 180,E1 -9311.8,E2 -9311.8} C_VEL
LIN {X 0,Y 432.331,Z 251.636,A -85,B 0,C 180,E1 -9314.347,E2 -9314.347} C_VEL
LIN {X 0,Y 432.3,Z 251.625,A -85,B 0,C 180,E1 -9317.018,E2 -9317.018} C_VEL
LIN {X 0,Y 432.286,Z 251.637,A -85,B 0,C 180,E1 -9319.827,E2 -9319.827} C_VEL
LIN {X 0,Y 432.293,Z 251.624,A -85,B 0,C 180,E1 -9323.02,E2 -9323.02} C_VEL
LIN {X 0,Y 432.356,Z 251.631,A -85,B 0,C 180,E1 -9325.996,E2 -9325.996} C_VEL
LIN {X 0,Y 432.342,Z 251.609,A -85,B 0,C 180,E1 -9329.489,E2 -9329.489} C_VEL
LIN {X 0,Y 432.323,Z 251.626,A -85,B 0,C 180,E1 -9331.872,E2 -9331.872} C_VEL
LIN {X 0,Y 432.371,Z 251.623,A -85,B 0,C 180,E1 -9335.539,E2 -9335.539} C_VEL
LIN {X 0,Y 432.344,Z 251.608,A -85,B 0,C 180,E1 -9339.045,E2 -9339.045} C_VEL
LIN {X 0,Y 432.366,Z 251.628,A -85,B 0,C 180,E1 -9342.01,E2 -9342.01} C_VEL
LIN {X 0,Y 432.386,Z 251.617,A -85,B 0,C 180,E1 -9344.926,E2 -9344.926} C_VEL
LIN {X 0,Y 432.452,Z 251.618,A -85,B 0,C 180,E1 -9347.803,E2 -9347.803} C_VEL
LIN {X 0,Y 432.455,Z 251.609,A -85,B 0,C 180,E1 -9351.589,E2 -9351.589} C_VEL
LIN {X 0,Y 432.544,Z 251.601,A -85,B 0,C 180,E1 -9354.405,E2 -9354.405} C_VEL
LIN {X 0,Y 432.587,Z 251.599,A -85,B 0,C 180,E1 -9358.138,E2 -9358.138} C_VEL
LIN {X 0,Y 432.611,Z 251.594,A -85,B 0,C 180,E1 -9360,E2 -9360} C_VEL
LIN {X 0,Y 432.56,Z 251.595,A -85,B 0,C 180,E1 -9362.794,E2 -9362.794} C_VEL
LIN {X 0,Y 432.499,Z 251.604,A -85,B 0,C 180,E1 -9366.531,E2 -9366.531} C_VEL
LIN {X 0,Y 432.429,Z 251.618,A -85,B 0,C 180,E1 -9369.353,E2 -9369.353} C_VEL
LIN {X 0,Y 432.424,Z 251.613,A -85,B 0,C 180,E1 -9372.803,E2 -9372.803} C_VEL
LIN {X 0,Y 432.404,Z 251.62,A -85,B 0,C 180,E1 -9376.478,E2 -9376.478} C_VEL
LIN {X 0,Y 432.331,Z 251.63,A -85,B 0,C 180,E1 -9379.961,E2 -9379.961} C_VEL
LIN {X 0,Y 432.303,Z 251.633,A -85,B 0,C 180,E1 -9382.965,E2 -9382.965} C_VEL
LIN {X 0,Y 432.31,Z 251.626,A -85,B 0,C 180,E1 -9386.036,E2 -9386.036} C_VEL
LIN {X 0,Y 432.315,Z 251.629,A -85,B 0,C 180,E1 -9389.189,E2 -9389.189} C_VEL
LIN {X 0,Y 432.311,Z 251.631,A -85,B 0,C 180,E1 -9392.444,E2 -9392.444} C_VEL
LIN {X 0,Y 432.328,Z 251.63,A -85,B 0,C 180,E1 -9395.819,E2 -9395.819} C_VEL
LIN {X 0,Y 432.295,Z 251.632,A -85,B 0,C 180,E1 -9399.349,E2 -9399.349} C_VEL
LIN {X 0,Y 432.298,Z 251.634,A -85,B 0,C 180,E1 -9401.801,E2 -9401.801} C_VEL
LIN {X 0,Y 432.33,Z 251.63,A -85,B 0,C 180,E1 -9404.348,E2 -9404.348} C_VEL
LIN {X 0,Y 432.297,Z 251.635,A -85,B 0,C 180,E1 -9407.019,E2 -9407.019} C_VEL
LIN {X 0,Y 432.285,Z 251.628,A -85,B 0,C 180,E1 -9409.829,E2 -9409.829} C_VEL
LIN {X 0,Y 432.291,Z 251.64,A -85,B 0,C 180,E1 -9413.021,E2 -9413.021} C_VEL
LIN {X 0,Y 432.33,Z 251.629,A -85,B 0,C 180,E1 -9416.002,E2 -9416.002} C_VEL
LIN {X 0,Y 432.351,Z 251.788,A -85,B 0,C 180,E1 -9419.14,E2 -9419.14} C_VEL
LIN {X 0,Y 435.507,Z 265.667,A -85,B 0,C 180,E1 -9421.572,E2 -9421.572} C_VEL
LIN {X 0,Y 436.414,Z 271.37,A -85,B 0,C 180,E1 -9422.514,E2 -9422.514} C_VEL
LIN {X 0,Y 435.292,Z 290.694,A -85,B 0,C 180,E1 -9425.434,E2 -9425.434} C_VEL
LIN {X 0,Y 434.286,Z 310.565,A -85,B 0,C 180,E1 -9428.398,E2 -9428.398} C_VEL
LIN {X 0,Y 433.444,Z 330.281,A -85,B 0,C 180,E1 -9431.264,E2 -9431.264} C_VEL
LIN {X 0,Y 436.604,Z 354.745,A -85,B 0,C 180,E1 -9431.847,E2 -9431.847} C_VEL
LIN {X 0,Y 437.464,Z 365.352,A -85,B 0,C 180,E1 -9432.069,E2 -9432.069} C_VEL
LIN {X 0,Y 436.634,Z 440.53,A -85,B 0,C 180,E1 -9433.339,E2 -9433.339} C_VEL
LIN {X 0,Y 436.047,Z 453.814,A -85,B 0,C 180,E1 -9433.737,E2 -9433.737} C_VEL
LIN {X 0,Y 435.266,Z 466.575,A -85,B 0,C 180,E1 -9434.309,E2 -9434.309} C_VEL
LIN {X 0,Y 434.612,Z 477.962,A -85,B 0,C 180,E1 -9435.005,E2 -9435.005} C_VEL
LIN {X 0,Y 433.771,Z 489.729,A -85,B 0,C 180,E1 -9435.934,E2 -9435.934} C_VEL
LIN {X 0,Y 433.169,Z 499.905,A -85,B 0,C 180,E1 -9436.941,E2 -9436.941} C_VEL
LIN {X 0,Y 432.487,Z 509.062,A -85,B 0,C 180,E1 -9438.042,E2 -9438.042} C_VEL
LIN {X 0,Y 432.088,Z 517.137,A -85,B 0,C 180,E1 -9439.219,E2 -9439.219} C_VEL
LIN {X 0,Y 431.723,Z 525.083,A -85,B 0,C 180,E1 -9440.631,E2 -9440.631} C_VEL
LIN {X 0,Y 431.562,Z 531.482,A -85,B 0,C 180,E1 -9442.043,E2 -9442.043} C_VEL
LIN {X 0,Y 431.497,Z 537.597,A -85,B 0,C 180,E1 -9443.771,E2 -9443.771} C_VEL
LIN {X 0,Y 431.525,Z 541.686,A -85,B 0,C 180,E1 -9445.329,E2 -9445.329} C_VEL
LIN {X 0,Y 431.644,Z 543.529,A -85,B 0,C 180,E1 -9446.266,E2 -9446.266} C_VEL
LIN {X 0,Y 431.638,Z 544.923,A -85,B 0,C 180,E1 -9447.2,E2 -9447.2} C_VEL
LIN {X 0,Y 431.631,Z 546.507,A -85,B 0,C 180,E1 -9449.067,E2 -9449.067} C_VEL
LIN {X 0,Y 431.674,Z 546.665,A -85,B 0,C 180,E1 -9450,E2 -9450} C_VEL
LIN {X 0,Y 431.644,Z 546.402,A -85,B 0,C 180,E1 -9450.933,E2 -9450.933} C_VEL
LIN {X 0,Y 431.649,Z 544.689,A -85,B 0,C 180,E1 -9452.799,E2 -9452.799} C_VEL
LIN {X 0,Y 431.732,Z 543.183,A -85,B 0,C 180,E1 -9453.733,E2 -9453.733} C_VEL
LIN {X 0,Y 431.529,Z 540.061,A -85,B 0,C 180,E1 -9455.139,E2 -9455.139} C_VEL
LIN {X 0,Y 431.563,Z 535.71,A -85,B 0,C 180,E1 -9456.593,E2 -9456.593} C_VEL
LIN {X 0,Y 431.581,Z 529.445,A -85,B 0,C 180,E1 -9458.191,E2 -9458.191} C_VEL
LIN {X 0,Y 431.771,Z 522.457,A -85,B 0,C 180,E1 -9459.604,E2 -9459.604} C_VEL
LIN {X 0,Y 432.135,Z 513.755,A -85,B 0,C 180,E1 -9461.016,E2 -9461.016} C_VEL
LIN {X 0,Y 432.628,Z 504.824,A -85,B 0,C 180,E1 -9462.191,E2 -9462.191} C_VEL
LIN {X 0,Y 433.191,Z 494.078,A -85,B 0,C 180,E1 -9463.342,E2 -9463.342} C_VEL
LIN {X 0,Y 433.772,Z 482.834,A -85,B 0,C 180,E1 -9464.304,E2 -9464.304} C_VEL
LIN {X 0,Y 434.543,Z 470.531,A -85,B 0,C 180,E1 -9465.116,E2 -9465.116} C_VEL
LIN {X 0,Y 435.221,Z 457.658,A -85,B 0,C 180,E1 -9465.752,E2 -9465.752} C_VEL
LIN {X 0,Y 435.741,Z 444.799,A -85,B 0,C 180,E1 -9466.183,E2 -9466.183} C_VEL
LIN {X 0,Y 435.938,Z 428.313,A -85,B 0,C 180,E1 -9466.507,E2 -9466.507} C_VEL
LIN {X 0,Y 436.388,Z 361.679,A -85,B 0,C 180,E1 -9467.597,E2 -9467.597} C_VEL
LIN {X 0,Y 433.108,Z 331.297,A -85,B 0,C 180,E1 -9468.232,E2 -9468.232} C_VEL
LIN {X 0,Y 433.128,Z 329.262,A -85,B 0,C 180,E1 -9468.445,E2 -9468.445} C_VEL
LIN {X 0,Y 433.799,Z 310.857,A -85,B 0,C 180,E1 -9471.128,E2 -9471.128} C_VEL
LIN {X 0,Y 434.794,Z 288.88,A -85,B 0,C 180,E1 -9474.341,E2 -9474.341} C_VEL
LIN {X 0,Y 435.732,Z 269.434,A -85,B 0,C 180,E1 -9477.211,E2 -9477.211} C_VEL
LIN {X 0,Y 433.752,Z 258.466,A -85,B 0,C 180,E1 -9478.961,E2 -9478.961} C_VEL
LIN {X 0,Y 432.35,Z 251.761,A -85,B 0,C 180,E1 -9480.09,E2 -9480.09} C_VEL
LIN {X 0,Y 432.308,Z 251.638,A -85,B 0,C 180,E1 -9483.554,E2 -9483.554} C_VEL
LIN {X 0,Y 432.326,Z 251.631,A -85,B 0,C 180,E1 -9485.817,E2 -9485.817} C_VEL
LIN {X 0,Y 432.305,Z 251.632,A -85,B 0,C 180,E1 -9488.708,E2 -9488.708} C_VEL
LIN {X 0,Y 432.294,Z 251.634,A -85,B 0,C 180,E1 -9491.8,E2 -9491.8} C_VEL
LIN {X 0,Y 432.324,Z 251.629,A -85,B 0,C 180,E1 -9494.347,E2 -9494.347} C_VEL
LIN {X 0,Y 432.292,Z 251.638,A -85,B 0,C 180,E1 -9497.018,E2 -9497.018} C_VEL
LIN {X 0,Y 432.279,Z 251.635,A -85,B 0,C 180,E1 -9499.827,E2 -9499.827} C_VEL
LIN {X 0,Y 432.287,Z 251.64,A -85,B 0,C 180,E1 -9503.02,E2 -9503.02} C_VEL
LIN {X 0,Y 432.32,Z 251.629,A -85,B 0,C 180,E1 -9506.002,E2 -9506.002} C_VEL
LIN {X 0,Y 432.326,Z 251.63,A -85,B 0,C 180,E1 -9509.491,E2 -9509.491} C_VEL
LIN {X 0,Y 432.302,Z 251.631,A -85,B 0,C 180,E1 -9511.871,E2 -9511.871} C_VEL
LIN {X 0,Y 432.335,Z 251.628,A -85,B 0,C 180,E1 -9515.547,E2 -9515.547} C_VEL
LIN {X 0,Y 432.333,Z 251.633,A -85,B 0,C 180,E1 -9519.045,E2 -9519.045} C_VEL
LIN {X 0,Y 432.343,Z 251.626,A -85,B 0,C 180,E1 -9522.01,E2 -9522.01} C_VEL
LIN {X 0,Y 432.366,Z 251.629,A -85,B 0,C 180,E1 -9524.926,E2 -9524.926} C_VEL
LIN {X 0,Y 432.445,Z 251.613,A -85,B 0,C 180,E1 -9527.803,E2 -9527.803} C_VEL
LIN {X 0,Y 432.434,Z 251.615,A -85,B 0,C 180,E1 -9531.589,E2 -9531.589} C_VEL
LIN {X 0,Y 432.531,Z 251.608,A -85,B 0,C 180,E1 -9534.405,E2 -9534.405} C_VEL
LIN {X 0,Y 432.585,Z 251.599,A -85,B 0,C 180,E1 -9538.138,E2 -9538.138} C_VEL
LIN {X 0,Y 432.532,Z 251.605,A -85,B 0,C 180,E1 -9540.931,E2 -9540.931} C_VEL
LIN {X 0,Y 432.541,Z 251.605,A -85,B 0,C 180,E1 -9542.794,E2 -9542.794} C_VEL
LIN {X 0,Y 432.501,Z 251.612,A -85,B 0,C 180,E1 -9546.532,E2 -9546.532} C_VEL
LIN {X 0,Y 432.404,Z 251.618,A -85,B 0,C 180,E1 -9549.354,E2 -9549.354} C_VEL
LIN {X 0,Y 432.419,Z 251.619,A -85,B 0,C 180,E1 -9552.803,E2 -9552.803} C_VEL
LIN {X 0,Y 432.399,Z 251.624,A -85,B 0,C 180,E1 -9556.478,E2 -9556.478} C_VEL
LIN {X 0,Y 432.326,Z 251.633,A -85,B 0,C 180,E1 -9559.961,E2 -9559.961} C_VEL
LIN {X 0,Y 432.299,Z 251.632,A -85,B 0,C 180,E1 -9562.966,E2 -9562.966} C_VEL
LIN {X 0,Y 432.306,Z 251.638,A -85,B 0,C 180,E1 -9566.037,E2 -9566.037} C_VEL
LIN {X 0,Y 432.313,Z 251.63,A -85,B 0,C 180,E1 -9569.19,E2 -9569.19} C_VEL
LIN {X 0,Y 432.308,Z 251.633,A -85,B 0,C 180,E1 -9572.445,E2 -9572.445} C_VEL
LIN {X 0,Y 432.324,Z 251.635,A -85,B 0,C 180,E1 -9575.82,E2 -9575.82} C_VEL
LIN {X 0,Y 432.291,Z 251.635,A -85,B 0,C 180,E1 -9579.35,E2 -9579.35} C_VEL
LIN {X 0,Y 432.293,Z 251.64,A -85,B 0,C 180,E1 -9581.802,E2 -9581.802} C_VEL
LIN {X 0,Y 432.326,Z 251.63,A -85,B 0,C 180,E1 -9584.349,E2 -9584.349} C_VEL
LIN {X 0,Y 432.295,Z 251.633,A -85,B 0,C 180,E1 -9587.02,E2 -9587.02} C_VEL
LIN {X 0,Y 432.283,Z 251.639,A -85,B 0,C 180,E1 -9589.829,E2 -9589.829} C_VEL
LIN {X 0,Y 432.291,Z 251.634,A -85,B 0,C 180,E1 -9593.022,E2 -9593.022} C_VEL
LIN {X 0,Y 432.327,Z 251.631,A -85,B 0,C 180,E1 -9596.004,E2 -9596.004} C_VEL
LIN {X 0,Y 432.329,Z 251.635,A -85,B 0,C 180,E1 -9599.495,E2 -9599.495} C_VEL
LIN {X 0,Y 432.311,Z 251.633,A -85,B 0,C 180,E1 -9601.873,E2 -9601.873} C_VEL
LIN {X 0,Y 432.315,Z 251.632,A -85,B 0,C 180,E1 -9604.998,E2 -9604.998} C_VEL
LIN {X 0,Y 432.353,Z 251.626,A -85,B 0,C 180,E1 -9608.046,E2 -9608.046} C_VEL
LIN {X 0,Y 432.346,Z 251.63,A -85,B 0,C 180,E1 -9611.029,E2 -9611.029} C_VEL
LIN {X 0,Y 432.362,Z 251.625,A -85,B 0,C 180,E1 -9613.959,E2 -9613.959} C_VEL
LIN {X 0,Y 432.452,Z 251.616,A -85,B 0,C 180,E1 -9617.804,E2 -9617.804} C_VEL
LIN {X 0,Y 432.43,Z 251.778,A -85,B 0,C 180,E1 -9620.026,E2 -9620.026} C_VEL
LIN {X 0,Y 432.655,Z 252.775,A -85,B 0,C 180,E1 -9620.185,E2 -9620.185} C_VEL
LIN {X 0,Y 437.154,Z 265.314,A -85,B 0,C 180,E1 -9620.587,E2 -9620.587} C_VEL
LIN {X 0,Y 436.436,Z 340.273,A -85,B 0,C 180,E1 -9621.842,E2 -9621.842} C_VEL
LIN {X 0,Y 436.361,Z 353.114,A -85,B 0,C 180,E1 -9622.248,E2 -9622.248} C_VEL
LIN {X 0,Y 436.094,Z 363.3,A -85,B 0,C 180,E1 -9622.705,E2 -9622.705} C_VEL
LIN {X 0,Y 435.527,Z 368.823,A -85,B 0,C 180,E1 -9622.993,E2 -9622.993} C_VEL
LIN {X 0,Y 432.501,Z 377.584,A -85,B 0,C 180,E1 -9623.461,E2 -9623.461} C_VEL
LIN {X 0,Y 429.177,Z 385.98,A -85,B 0,C 180,E1 -9624.01,E2 -9624.01} C_VEL
LIN {X 0,Y 428.144,Z 390.853,A -85,B 0,C 180,E1 -9624.421,E2 -9624.421} C_VEL
LIN {X 0,Y 427.578,Z 401.197,A -85,B 0,C 180,E1 -9625.523,E2 -9625.523} C_VEL
LIN {X 0,Y 426.997,Z 410.122,A -85,B 0,C 180,E1 -9626.698,E2 -9626.698} C_VEL
LIN {X 0,Y 426.45,Z 418.817,A -85,B 0,C 180,E1 -9628.112,E2 -9628.112} C_VEL
LIN {X 0,Y 425.899,Z 425.834,A -85,B 0,C 180,E1 -9629.528,E2 -9629.528} C_VEL
LIN {X 0,Y 425.524,Z 431.42,A -85,B 0,C 180,E1 -9630.947,E2 -9630.947} C_VEL
LIN {X 0,Y 425.305,Z 435.817,A -85,B 0,C 180,E1 -9632.368,E2 -9632.368} C_VEL
LIN {X 0,Y 425.056,Z 439.182,A -85,B 0,C 180,E1 -9633.792,E2 -9633.792} C_VEL
LIN {X 0,Y 425.077,Z 440.836,A -85,B 0,C 180,E1 -9634.742,E2 -9634.742} C_VEL
LIN {X 0,Y 425.026,Z 442.113,A -85,B 0,C 180,E1 -9635.694,E2 -9635.694} C_VEL
LIN {X 0,Y 424.95,Z 443.277,A -85,B 0,C 180,E1 -9637.108,E2 -9637.108} C_VEL
LIN {X 0,Y 424.936,Z 443.579,A -85,B 0,C 180,E1 -9638.561,E2 -9638.561} C_VEL
LIN {X 0,Y 425.025,Z 442.603,A -85,B 0,C 180,E1 -9640.48,E2 -9640.48} C_VEL
LIN {X 0,Y 425.098,Z 441.494,A -85,B 0,C 180,E1 -9641.443,E2 -9641.443} C_VEL
LIN {X 0,Y 425.354,Z 439.075,A -85,B 0,C 180,E1 -9642.877,E2 -9642.877} C_VEL
LIN {X 0,Y 425.659,Z 435.592,A -85,B 0,C 180,E1 -9644.339,E2 -9644.339} C_VEL
LIN {X 0,Y 426.054,Z 431.001,A -85,B 0,C 180,E1 -9645.794,E2 -9645.794} C_VEL
LIN {X 0,Y 426.647,Z 424.015,A -85,B 0,C 180,E1 -9647.495,E2 -9647.495} C_VEL
LIN {X 0,Y 427.323,Z 416.365,A -85,B 0,C 180,E1 -9648.955,E2 -9648.955} C_VEL
LIN {X 0,Y 428.06,Z 407.174,A -85,B 0,C 180,E1 -9650.347,E2 -9650.347} C_VEL
LIN {X 0,Y 428.708,Z 397.645,A -85,B 0,C 180,E1 -9651.518,E2 -9651.518} C_VEL
LIN {X 0,Y 429.383,Z 387.817,A -85,B 0,C 180,E1 -9652.494,E2 -9652.494} C_VEL
LIN {X 0,Y 430.002,Z 377.141,A -85,B 0,C 180,E1 -9653.343,E2 -9653.343} C_VEL
LIN {X 0,Y 430.431,Z 366.208,A -85,B 0,C 180,E1 -9654.029,E2 -9654.029} C_VEL
LIN {X 0,Y 430.728,Z 353.218,A -85,B 0,C 180,E1 -9654.635,E2 -9654.635} C_VEL
LIN {X 0,Y 430.889,Z 341.779,A -85,B 0,C 180,E1 -9654.995,E2 -9654.995} C_VEL
LIN {X 0,Y 431.183,Z 305.814,A -85,B 0,C 180,E1 -9655.636,E2 -9655.636} C_VEL
LIN {X 0,Y 431.584,Z 268.046,A -85,B 0,C 180,E1 -9656.278,E2 -9656.278} C_VEL
LIN {X 0,Y 425.49,Z 253.557,A -85,B 0,C 180,E1 -9656.881,E2 -9656.881} C_VEL
LIN {X 0,Y 425.317,Z 252.656,A -85,B 0,C 180,E1 -9657.043,E2 -9657.043} C_VEL
LIN {X 0,Y 425.285,Z 252.502,A -85,B 0,C 180,E1 -9659.72,E2 -9659.72} C_VEL
LIN {X 0,Y 425.271,Z 252.512,A -85,B 0,C 180,E1 -9663.049,E2 -9663.049} C_VEL
LIN {X 0,Y 425.28,Z 252.481,A -85,B 0,C 180,E1 -9665.927,E2 -9665.927} C_VEL
LIN {X 0,Y 425.26,Z 252.512,A -85,B 0,C 180,E1 -9669.036,E2 -9669.036} C_VEL
LIN {X 0,Y 425.257,Z 252.507,A -85,B 0,C 180,E1 -9672.655,E2 -9672.655} C_VEL
LIN {X 0,Y 425.282,Z 252.507,A -85,B 0,C 180,E1 -9675.283,E2 -9675.283} C_VEL
LIN {X 0,Y 425.245,Z 252.514,A -85,B 0,C 180,E1 -9678.617,E2 -9678.617} C_VEL
LIN {X 0,Y 425.273,Z 252.502,A -85,B 0,C 180,E1 -9681.098,E2 -9681.098} C_VEL
LIN {X 0,Y 425.293,Z 252.509,A -85,B 0,C 180,E1 -9684.663,E2 -9684.663} C_VEL
LIN {X 0,Y 425.261,Z 252.502,A -85,B 0,C 180,E1 -9688.072,E2 -9688.072} C_VEL
LIN {X 0,Y 425.301,Z 252.497,A -85,B 0,C 180,E1 -9691.365,E2 -9691.365} C_VEL
LIN {X 0,Y 425.262,Z 252.51,A -85,B 0,C 180,E1 -9694.552,E2 -9694.552} C_VEL
LIN {X 0,Y 425.278,Z 252.492,A -85,B 0,C 180,E1 -9696.633,E2 -9696.633} C_VEL
LIN {X 0,Y 425.289,Z 252.489,A -85,B 0,C 180,E1 -9699.694,E2 -9699.694} C_VEL
LIN {X 0,Y 425.333,Z 252.502,A -85,B 0,C 180,E1 -9702.697,E2 -9702.697} C_VEL
LIN {X 0,Y 425.339,Z 252.496,A -85,B 0,C 180,E1 -9705.649,E2 -9705.649} C_VEL
LIN {X 0,Y 425.341,Z 252.499,A -85,B 0,C 180,E1 -9708.563,E2 -9708.563} C_VEL
LIN {X 0,Y 425.399,Z 252.486,A -85,B 0,C 180,E1 -9711.449,E2 -9711.449} C_VEL
LIN {X 0,Y 425.502,Z 252.479,A -85,B 0,C 180,E1 -9714.312,E2 -9714.312} C_VEL
LIN {X 0,Y 425.556,Z 252.476,A -85,B 0,C 180,E1 -9718.107,E2 -9718.107} C_VEL
LIN {X 0,Y 425.564,Z 252.472,A -85,B 0,C 180,E1 -9720,E2 -9720} C_VEL
LIN {X 0,Y 425.516,Z 252.472,A -85,B 0,C 180,E1 -9722.84,E2 -9722.84} C_VEL
LIN {X 0,Y 425.462,Z 252.48,A -85,B 0,C 180,E1 -9726.64,E2 -9726.64} C_VEL
LIN {X 0,Y 425.388,Z 252.497,A -85,B 0,C 180,E1 -9729.51,E2 -9729.51} C_VEL
LIN {X 0,Y 425.387,Z 252.49,A -85,B 0,C 180,E1 -9732.903,E2 -9732.903} C_VEL
LIN {X 0,Y 425.353,Z 252.498,A -85,B 0,C 180,E1 -9736.604,E2 -9736.604} C_VEL
LIN {X 0,Y 425.322,Z 252.506,A -85,B 0,C 180,E1 -9739.635,E2 -9739.635} C_VEL
LIN {X 0,Y 425.281,Z 252.504,A -85,B 0,C 180,E1 -9742.339,E2 -9742.339} C_VEL
LIN {X 0,Y 425.252,Z 252.509,A -85,B 0,C 180,E1 -9745.448,E2 -9745.448} C_VEL
LIN {X 0,Y 425.293,Z 252.498,A -85,B 0,C 180,E1 -9748.858,E2 -9748.858} C_VEL
LIN {X 0,Y 425.249,Z 252.51,A -85,B 0,C 180,E1 -9751.928,E2 -9751.928} C_VEL
LIN {X 0,Y 425.287,Z 252.51,A -85,B 0,C 180,E1 -9755.337,E2 -9755.337} C_VEL
LIN {X 0,Y 425.271,Z 252.505,A -85,B 0,C 180,E1 -9758.902,E2 -9758.902} C_VEL
LIN {X 0,Y 425.251,Z 252.511,A -85,B 0,C 180,E1 -9762.656,E2 -9762.656} C_VEL
LIN {X 0,Y 425.28,Z 252.509,A -85,B 0,C 180,E1 -9765.284,E2 -9765.284} C_VEL
LIN {X 0,Y 425.243,Z 252.516,A -85,B 0,C 180,E1 -9768.618,E2 -9768.618} C_VEL
LIN {X 0,Y 425.27,Z 252.496,A -85,B 0,C 180,E1 -9771.099,E2 -9771.099} C_VEL
LIN {X 0,Y 425.289,Z 252.498,A -85,B 0,C 180,E1 -9774.664,E2 -9774.664} C_VEL
LIN {X 0,Y 425.254,Z 252.504,A -85,B 0,C 180,E1 -9778.073,E2 -9778.073} C_VEL
LIN {X 0,Y 425.314,Z 252.731,A -85,B 0,C 180,E1 -9778.842,E2 -9778.842} C_VEL
LIN {X 0,Y 428.9,Z 268.423,A -85,B 0,C 180,E1 -9781.628,E2 -9781.628} C_VEL
LIN {X 0,Y 429.532,Z 272.301,A -85,B 0,C 180,E1 -9782.281,E2 -9782.281} C_VEL
LIN {X 0,Y 428.492,Z 290.081,A -85,B 0,C 180,E1 -9785.018,E2 -9785.018} C_VEL
LIN {X 0,Y 427.328,Z 311.588,A -85,B 0,C 180,E1 -9788.282,E2 -9788.282} C_VEL
LIN {X 0,Y 426.519,Z 329.166,A -85,B 0,C 180,E1 -9790.897,E2 -9790.897} C_VEL
LIN {X 0,Y 429.948,Z 355.707,A -85,B 0,C 180,E1 -9791.548,E2 -9791.548} C_VEL
LIN {X 0,Y 430.764,Z 366.761,A -85,B 0,C 180,E1 -9791.781,E2 -9791.781} C_VEL
LIN {X 0,Y 429.895,Z 439.893,A -85,B 0,C 180,E1 -9793.039,E2 -9793.039} C_VEL
LIN {X 0,Y 429.296,Z 453.095,A -85,B 0,C 180,E1 -9793.444,E2 -9793.444} C_VEL
LIN {X 0,Y 428.452,Z 466.373,A -85,B 0,C 180,E1 -9794.053,E2 -9794.053} C_VEL
LIN {X 0,Y 427.757,Z 477.57,A -85,B 0,C 180,E1 -9794.759,E2 -9794.759} C_VEL
LIN {X 0,Y 426.848,Z 489.238,A -85,B 0,C 180,E1 -9795.701,E2 -9795.701} C_VEL
LIN {X 0,Y 426.14,Z 500.344,A -85,B 0,C 180,E1 -9796.834,E2 -9796.834} C_VEL
LIN {X 0,Y 425.504,Z 508.449,A -85,B 0,C 180,E1 -9797.843,E2 -9797.843} C_VEL
LIN {X 0,Y 425.072,Z 516.479,A -85,B 0,C 180,E1 -9799.039,E2 -9799.039} C_VEL
LIN {X 0,Y 424.676,Z 524.371,A -85,B 0,C 180,E1 -9800.474,E2 -9800.474} C_VEL
LIN {X 0,Y 424.495,Z 530.74,A -85,B 0,C 180,E1 -9801.91,E2 -9801.91} C_VEL
LIN {X 0,Y 424.456,Z 536.149,A -85,B 0,C 180,E1 -9803.445,E2 -9803.445} C_VEL
LIN {X 0,Y 424.424,Z 539.79,A -85,B 0,C 180,E1 -9804.774,E2 -9804.774} C_VEL
LIN {X 0,Y 424.57,Z 542.72,A -85,B 0,C 180,E1 -9806.203,E2 -9806.203} C_VEL
LIN {X 0,Y 424.586,Z 544.107,A -85,B 0,C 180,E1 -9807.153,E2 -9807.153} C_VEL
LIN {X 0,Y 424.578,Z 545.668,A -85,B 0,C 180,E1 -9809.051,E2 -9809.051} C_VEL
LIN {X 0,Y 424.626,Z 545.81,A -85,B 0,C 180,E1 -9810,E2 -9810} C_VEL
LIN {X 0,Y 424.594,Z 545.537,A -85,B 0,C 180,E1 -9810.948,E2 -9810.948} C_VEL
LIN {X 0,Y 424.573,Z 544.868,A -85,B 0,C 180,E1 -9811.897,E2 -9811.897} C_VEL
LIN {X 0,Y 424.6,Z 543.802,A -85,B 0,C 180,E1 -9812.846,E2 -9812.846} C_VEL
LIN {X 0,Y 424.654,Z 542.273,A -85,B 0,C 180,E1 -9813.795,E2 -9813.795} C_VEL
LIN {X 0,Y 424.463,Z 539.128,A -85,B 0,C 180,E1 -9815.224,E2 -9815.224} C_VEL
LIN {X 0,Y 424.499,Z 534.918,A -85,B 0,C 180,E1 -9816.655,E2 -9816.655} C_VEL
LIN {X 0,Y 424.526,Z 528.455,A -85,B 0,C 180,E1 -9818.328,E2 -9818.328} C_VEL
LIN {X 0,Y 424.717,Z 521.431,A -85,B 0,C 180,E1 -9819.765,E2 -9819.765} C_VEL
LIN {X 0,Y 425.113,Z 512.672,A -85,B 0,C 180,E1 -9821.2,E2 -9821.2} C_VEL
LIN {X 0,Y 425.656,Z 503.697,A -85,B 0,C 180,E1 -9822.394,E2 -9822.394} C_VEL
LIN {X 0,Y 426.177,Z 493.842,A -85,B 0,C 180,E1 -9823.469,E2 -9823.469} C_VEL
LIN {X 0,Y 426.746,Z 483.075,A -85,B 0,C 180,E1 -9824.423,E2 -9824.423} C_VEL
LIN {X 0,Y 427.54,Z 471.112,A -85,B 0,C 180,E1 -9825.248,E2 -9825.248} C_VEL
LIN {X 0,Y 428.238,Z 458.676,A -85,B 0,C 180,E1 -9825.894,E2 -9825.894} C_VEL
LIN {X 0,Y 428.803,Z 445.932,A -85,B 0,C 180,E1 -9826.361,E2 -9826.361} C_VEL
LIN {X 0,Y 429.034,Z 432.571,A -85,B 0,C 180,E1 -9826.658,E2 -9826.658} C_VEL
LIN {X 0,Y 429.519,Z 361.926,A -85,B 0,C 180,E1 -9827.831,E2 -9827.831} C_VEL
LIN {X 0,Y 426.098,Z 330.145,A -85,B 0,C 180,E1 -9828.511,E2 -9828.511} C_VEL
LIN {X 0,Y 426.405,Z 321.836,A -85,B 0,C 180,E1 -9829.691,E2 -9829.691} C_VEL
LIN {X 0,Y 427.586,Z 294.525,A -85,B 0,C 180,E1 -9833.746,E2 -9833.746} C_VEL
LIN {X 0,Y 428.687,Z 272.387,A -85,B 0,C 180,E1 -9837.06,E2 -9837.06} C_VEL
LIN {X 0,Y 428.52,Z 268.445,A -85,B 0,C 180,E1 -9837.67,E2 -9837.67} C_VEL
LIN {X 0,Y 425.319,Z 252.682,A -85,B 0,C 180,E1 -9840.293,E2 -9840.293} C_VEL
LIN {X 0,Y 425.262,Z 252.513,A -85,B 0,C 180,E1 -9843.048,E2 -9843.048} C_VEL
LIN {X 0,Y 425.27,Z 252.509,A -85,B 0,C 180,E1 -9845.926,E2 -9845.926} C_VEL
LIN {X 0,Y 425.237,Z 252.515,A -85,B 0,C 180,E1 -9849.033,E2 -9849.033} C_VEL
LIN {X 0,Y 425.247,Z 252.511,A -85,B 0,C 180,E1 -9852.655,E2 -9852.655} C_VEL
LIN {X 0,Y 425.277,Z 252.514,A -85,B 0,C 180,E1 -9855.282,E2 -9855.282} C_VEL
LIN {X 0,Y 425.238,Z 252.513,A -85,B 0,C 180,E1 -9858.617,E2 -9858.617} C_VEL
LIN {X 0,Y 425.268,Z 252.515,A -85,B 0,C 180,E1 -9861.098,E2 -9861.098} C_VEL
LIN {X 0,Y 425.281,Z 252.508,A -85,B 0,C 180,E1 -9864.662,E2 -9864.662} C_VEL
LIN {X 0,Y 425.235,Z 252.512,A -85,B 0,C 180,E1 -9868.071,E2 -9868.071} C_VEL
LIN {X 0,Y 425.283,Z 252.509,A -85,B 0,C 180,E1 -9871.364,E2 -9871.364} C_VEL
LIN {X 0,Y 425.239,Z 252.514,A -85,B 0,C 180,E1 -9874.551,E2 -9874.551} C_VEL
LIN {X 0,Y 425.28,Z 252.506,A -85,B 0,C 180,E1 -9877.73,E2 -9877.73} C_VEL
LIN {X 0,Y 425.348,Z 252.504,A -85,B 0,C 180,E1 -9880.703,E2 -9880.703} C_VEL
LIN {X 0,Y 425.371,Z 252.495,A -85,B 0,C 180,E1 -9883.688,E2 -9883.688} C_VEL
LIN {X 0,Y 425.399,Z 252.491,A -85,B 0,C 180,E1 -9887.598,E2 -9887.598} C_VEL
LIN {X 0,Y 425.382,Z 252.494,A -85,B 0,C 180,E1 -9891.449,E2 -9891.449} C_VEL
LIN {X 0,Y 425.489,Z 252.484,A -85,B 0,C 180,E1 -9894.313,E2 -9894.313} C_VEL
LIN {X 0,Y 425.554,Z 252.474,A -85,B 0,C 180,E1 -9898.107,E2 -9898.107} C_VEL
LIN {X 0,Y 425.494,Z 252.482,A -85,B 0,C 180,E1 -9900.947,E2 -9900.947} C_VEL
LIN {X 0,Y 425.496,Z 252.482,A -85,B 0,C 180,E1 -9902.84,E2 -9902.84} C_VEL
LIN {X 0,Y 425.462,Z 252.488,A -85,B 0,C 180,E1 -9906.615,E2 -9906.615} C_VEL
LIN {X 0,Y 425.366,Z 252.496,A -85,B 0,C 180,E1 -9909.51,E2 -9909.51} C_VEL
LIN {X 0,Y 425.381,Z 252.495,A -85,B 0,C 180,E1 -9912.903,E2 -9912.903} C_VEL
LIN {X 0,Y 425.348,Z 252.501,A -85,B 0,C 180,E1 -9916.604,E2 -9916.604} C_VEL
LIN {X 0,Y 425.317,Z 252.503,A -85,B 0,C 180,E1 -9919.636,E2 -9919.636} C_VEL
LIN {X 0,Y 425.277,Z 252.511,A -85,B 0,C 180,E1 -9922.34,E2 -9922.34} C_VEL
LIN {X 0,Y 425.247,Z 252.511,A -85,B 0,C 180,E1 -9925.449,E2 -9925.449} C_VEL
LIN {X 0,Y 425.291,Z 252.505,A -85,B 0,C 180,E1 -9928.859,E2 -9928.859} C_VEL
LIN {X 0,Y 425.251,Z 252.517,A -85,B 0,C 180,E1 -9931.929,E2 -9931.929} C_VEL
LIN {X 0,Y 425.283,Z 252.507,A -85,B 0,C 180,E1 -9935.338,E2 -9935.338} C_VEL
LIN {X 0,Y 425.265,Z 252.508,A -85,B 0,C 180,E1 -9938.903,E2 -9938.903} C_VEL
LIN {X 0,Y 425.248,Z 252.51,A -85,B 0,C 180,E1 -9942.657,E2 -9942.657} C_VEL
LIN {X 0,Y 425.278,Z 252.508,A -85,B 0,C 180,E1 -9945.285,E2 -9945.285} C_VEL
LIN {X 0,Y 425.24,Z 252.511,A -85,B 0,C 180,E1 -9948.619,E2 -9948.619} C_VEL
LIN {X 0,Y 425.269,Z 252.509,A -85,B 0,C 180,E1 -9951.1,E2 -9951.1} C_VEL
LIN {X 0,Y 425.286,Z 252.505,A -85,B 0,C 180,E1 -9954.664,E2 -9954.664} C_VEL
LIN {X 0,Y 425.244,Z 252.512,A -85,B 0,C 180,E1 -9958.073,E2 -9958.073} C_VEL
LIN {X 0,Y 425.291,Z 252.511,A -85,B 0,C 180,E1 -9961.366,E2 -9961.366} C_VEL
LIN {X 0,Y 425.25,Z 252.51,A -85,B 0,C 180,E1 -9964.553,E2 -9964.553} C_VEL
LIN {X 0,Y 425.291,Z 252.508,A -85,B 0,C 180,E1 -9967.732,E2 -9967.732} C_VEL
LIN {X 0,Y 425.326,Z 252.501,A -85,B 0,C 180,E1 -9970.703,E2 -9970.703} C_VEL
LIN {X 0,Y 425.315,Z 252.504,A -85,B 0,C 180,E1 -9973.686,E2 -9973.686} C_VEL
LIN {X 0,Y 425.405,Z 252.496,A -85,B 0,C 180,E1 -9977.599,E2 -9977.599} C_VEL
LIN {X 0,Y 425.36,Z 252.68,A -85,B 0,C 180,E1 -9979.769,E2 -9979.769} C_VEL
LIN {X 0,Y 425.595,Z 253.66,A -85,B 0,C 180,E1 -9979.923,E2 -9979.923} C_VEL
LIN {X 0,Y 430.414,Z 267.149,A -85,B 0,C 180,E1 -9980.36,E2 -9980.36} C_VEL
LIN {X 0,Y 429.601,Z 340.317,A -85,B 0,C 180,E1 -9981.593,E2 -9981.593} C_VEL
LIN {X 0,Y 429.491,Z 353.445,A -85,B 0,C 180,E1 -9982.005,E2 -9982.005} C_VEL
LIN {X 0,Y 429.208,Z 364.938,A -85,B 0,C 180,E1 -9982.533,E2 -9982.533} C_VEL
LIN {X 0,Y 428.824,Z 377.256,A -85,B 0,C 180,E1 -9983.295,E2 -9983.295} C_VEL
LIN {X 0,Y 428.253,Z 388.806,A -85,B 0,C 180,E1 -9984.232,E2 -9984.232} C_VEL
LIN {X 0,Y 428.144,Z 390.853,A -85,B 0,C 180,E1 -9984.421,E2 -9984.421} C_VEL
LIN {X 0,Y 427.156,Z 395.669,A -85,B 0,C 180,E1 -9984.865,E2 -9984.865} C_VEL
LIN {X 0,Y 423.911,Z 403.237,A -85,B 0,C 180,E1 -9985.614,E2 -9985.614} C_VEL
LIN {X 0,Y 420.722,Z 410.255,A -85,B 0,C 180,E1 -9986.458,E2 -9986.458} C_VEL
LIN {X 0,Y 419.828,Z 414.206,A -85,B 0,C 180,E1 -9987.043,E2 -9987.043} C_VEL
LIN {X 0,Y 419.259,Z 422.645,A -85,B 0,C 180,E1 -9988.56,E2 -9988.56} C_VEL
LIN {X 0,Y 418.793,Z 429.057,A -85,B 0,C 180,E1 -9990,E2 -9990} C_VEL
LIN {X 0,Y 418.451,Z 434.162,A -85,B 0,C 180,E1 -9991.444,E2 -9991.444} C_VEL
LIN {X 0,Y 418.138,Z 438.143,A -85,B 0,C 180,E1 -9992.891,E2 -9992.891} C_VEL
LIN {X 0,Y 418.01,Z 440.209,A -85,B 0,C 180,E1 -9993.856,E2 -9993.856} C_VEL
LIN {X 0,Y 418.045,Z 441.829,A -85,B 0,C 180,E1 -9994.822,E2 -9994.822} C_VEL
LIN {X 0,Y 417.988,Z 443.075,A -85,B 0,C 180,E1 -9995.79,E2 -9995.79} C_VEL
LIN {X 0,Y 417.91,Z 444.139,A -85,B 0,C 180,E1 -9997.155,E2 -9997.155} C_VEL
LIN {X 0,Y 417.891,Z 444.416,A -85,B 0,C 180,E1 -9998.706,E2 -9998.706} C_VEL
LIN {X 0,Y 417.95,Z 444.084,A -85,B 0,C 180,E1 -9999.681,E2 -9999.681} C_VEL
LIN {X 0,Y 418.011,Z 443.363,A -85,B 0,C 180,E1 -10000.658,E2 -10000.658} C_VEL
LIN {X 0,Y 418.105,Z 442.199,A -85,B 0,C 180,E1 -10001.637,E2 -10001.637} C_VEL
LIN {X 0,Y 418.374,Z 439.885,A -85,B 0,C 180,E1 -10003.014,E2 -10003.014} C_VEL
LIN {X 0,Y 418.716,Z 436.156,A -85,B 0,C 180,E1 -10004.582,E2 -10004.582} C_VEL
LIN {X 0,Y 419.148,Z 431.487,A -85,B 0,C 180,E1 -10006.061,E2 -10006.061} C_VEL
LIN {X 0,Y 419.669,Z 425.529,A -85,B 0,C 180,E1 -10007.544,E2 -10007.544} C_VEL
LIN {X 0,Y 420.396,Z 418.048,A -85,B 0,C 180,E1 -10009.026,E2 -10009.026} C_VEL
LIN {X 0,Y 421.055,Z 410.349,A -85,B 0,C 180,E1 -10010.264,E2 -10010.264} C_VEL
LIN {X 0,Y 421.782,Z 400.861,A -85,B 0,C 180,E1 -10011.505,E2 -10011.505} C_VEL
LIN {X 0,Y 422.519,Z 390.234,A -85,B 0,C 180,E1 -10012.622,E2 -10012.622} C_VEL
LIN {X 0,Y 423.141,Z 379.913,A -85,B 0,C 180,E1 -10013.492,E2 -10013.492} C_VEL
LIN {X 0,Y 423.706,Z 369.013,A -85,B 0,C 180,E1 -10014.217,E2 -10014.217} C_VEL
LIN {X 0,Y 424.049,Z 356.64,A -85,B 0,C 180,E1 -10014.837,E2 -10014.837} C_VEL
LIN {X 0,Y 424.208,Z 344.714,A -85,B 0,C 180,E1 -10015.252,E2 -10015.252} C_VEL
LIN {X 0,Y 424.284,Z 326.532,A -85,B 0,C 180,E1 -10015.62,E2 -10015.62} C_VEL
LIN {X 0,Y 425.003,Z 269.894,A -85,B 0,C 180,E1 -10016.591,E2 -10016.591} C_VEL
LIN {X 0,Y 418.427,Z 254.336,A -85,B 0,C 180,E1 -10017.264,E2 -10017.264} C_VEL
LIN {X 0,Y 418.246,Z 253.474,A -85,B 0,C 180,E1 -10017.455,E2 -10017.455} C_VEL
LIN {X 0,Y 418.243,Z 253.369,A -85,B 0,C 180,E1 -10020.272,E2 -10020.272} C_VEL
LIN {X 0,Y 418.234,Z 253.389,A -85,B 0,C 180,E1 -10023.678,E2 -10023.678} C_VEL
LIN {X 0,Y 418.237,Z 253.359,A -85,B 0,C 180,E1 -10027.224,E2 -10027.224} C_VEL
LIN {X 0,Y 418.207,Z 253.388,A -85,B 0,C 180,E1 -10030.866,E2 -10030.866} C_VEL
LIN {X 0,Y 418.201,Z 253.391,A -85,B 0,C 180,E1 -10033.727,E2 -10033.727} C_VEL
LIN {X 0,Y 418.197,Z 253.381,A -85,B 0,C 180,E1 -10036.446,E2 -10036.446} C_VEL
LIN {X 0,Y 418.205,Z 253.39,A -85,B 0,C 180,E1 -10039.132,E2 -10039.132} C_VEL
LIN {X 0,Y 418.23,Z 253.372,A -85,B 0,C 180,E1 -10042.774,E2 -10042.774} C_VEL
LIN {X 0,Y 418.245,Z 253.389,A -85,B 0,C 180,E1 -10046.322,E2 -10046.322} C_VEL
LIN {X 0,Y 418.238,Z 253.364,A -85,B 0,C 180,E1 -10049.727,E2 -10049.727} C_VEL
LIN {X 0,Y 418.207,Z 253.39,A -85,B 0,C 180,E1 -10053.016,E2 -10053.016} C_VEL
LIN {X 0,Y 418.268,Z 253.369,A -85,B 0,C 180,E1 -10056.217,E2 -10056.217} C_VEL
LIN {X 0,Y 418.244,Z 253.363,A -85,B 0,C 180,E1 -10059.336,E2 -10059.336} C_VEL
LIN {X 0,Y 418.279,Z 253.382,A -85,B 0,C 180,E1 -10062.396,E2 -10062.396} C_VEL
LIN {X 0,Y 418.294,Z 253.373,A -85,B 0,C 180,E1 -10065.402,E2 -10065.402} C_VEL
LIN {X 0,Y 418.306,Z 253.377,A -85,B 0,C 180,E1 -10068.368,E2 -10068.368} C_VEL
LIN {X 0,Y 418.44,Z 253.361,A -85,B 0,C 180,E1 -10072.278,E2 -10072.278} C_VEL
LIN {X 0,Y 418.463,Z 253.356,A -85,B 0,C 180,E1 -10074.216,E2 -10074.216} C_VEL
LIN {X 0,Y 418.525,Z 253.352,A -85,B 0,C 180,E1 -10078.075,E2 -10078.075} C_VEL
LIN {X 0,Y 418.399,Z 253.362,A -85,B 0,C 180,E1 -10080.962,E2 -10080.962} C_VEL
LIN {X 0,Y 418.473,Z 253.35,A -85,B 0,C 180,E1 -10082.888,E2 -10082.888} C_VEL
LIN {X 0,Y 418.428,Z 253.357,A -85,B 0,C 180,E1 -10086.752,E2 -10086.752} C_VEL
